(* CODESYS project Piezo.library
   Company: ESO
   Description: Local Device Control - LDC Piezo Library based on State Machine
   Version: 0.6.6.3
   Placeholder: ESO LDC Piezo Library
   Author: Dan Popovic
   Title: ESO LDC Piezo Library

Project tree, tasks and I/O mapping:
  libraries: Tc2_Standard, * (Beckhoff Automation GmbH); Tc2_System, * (Beckhoff Automation GmbH); Tc2_Utilities, * (Beckhoff Automation GmbH); Tc3_EventLogger, * (Beckhoff Automation GmbH); Tc3_Module, * (Beckhoff Automation GmbH); VisuDialogs, * (System); VisuSymbols, 3.5.10.0 (System)
  config/
    Device1_EtherCAT_SPLC014.xti
    Mappings_HW_SPLC014.xml
    Mappings_SIM.xml
  00000000-0000-0000-0000-000000000000|config\Device1_EtherCAT_SPLC014.xti
  00000000-0000-0000-0000-000000000000|config\Mappings_HW_SPLC014.xml
  00000000-0000-0000-0000-000000000000|config\Mappings_SIM.xml
  doc/
  DUTs/
    Enumerated/
      data type E_PIEZO_COMMAND
      data type E_PIEZO_ERROR
      data type E_PIEZO_EVENT
      data type E_PIEZO_HW_STATUS
      data type E_PIEZO_RPC_ERROR
      data type E_PIEZO_STATE
      data type E_PIEZO_STATUS
      data type E_PIEZO_SUBSTATE
    Structures/
      data type T_PIEZO_CFG
      data type T_PIEZO_CTRL
      data type T_PIEZO_DINT
      data type T_PIEZO_INFO
      data type T_PIEZO_INT
      data type T_PIEZO_LREAL
      data type T_PIEZO_STAT
      data type T_SIM_PIEZO_CFG
  GVLs/
    global variables GVL
  lib/
  POUs/
    Examples/
      function block FB_PIEZO_EXAMPLE [ST]: ActivityAuto, ActivityPos, M_Configure
    function block FB_PIEZO_BASE [ST]: ActionAutoExecute, ActionDisableExecute, ActionEnableExecute, ActionErrExecute, ActionHomeExecute, ActionInitExecute, ActionMaxOnFailure, ActionMoveBitExecute, ActionMoveUserExecute, ActionPosExecute, ActionResetExecute, ActionStopExecute, ActivityAuto, ActivityPos, CheckForEvents, M_CheckMaxOn, M_CheckRangeBit, M_CheckRangeUser, M_Configure, M_GetLogicalState, M_GetRpcErrorText, M_GetTimeInSec, M_LogEventDebug, M_LogEventEnd, M_LogEventError, M_LogEventGeneral, M_LogEventStart, M_ResetOutputs, M_RestartMaxOnTimer, M_SetRpcStatus, M_UpdateMonitor, ProcessEvents, RPC_Auto, RPC_Disable, RPC_Enable, RPC_Home, RPC_Init, RPC_MoveBit, RPC_MoveUser, RPC_Pos, RPC_Reset, RPC_SetDebug, RPC_SetLog, RPC_Stop, SetAction, SetEvent, SetHwStatus, SetLastCommand, SetState, SetStatus
    function block FB_SIM_PIEZO [ST]: RPC_ResetConfig, RPC_SetCouplerState, RPC_SetMaxError
    program MAIN [ST]
  Version/
    global variables Global_Version
  VISUs/
    Templates/
      visualisation GUI_TEMPLATE_PIEZO
    visualisation GUI_Piezo001
    visualisation GUI_Piezo002
  text list GlobalTextList
  00000000-0000-0000-0000-000000000000|Piezo.tmc
  Piezo.tmc
*)

// DUTs/Enumerated/E_PIEZO_COMMAND
{attribute 'qualified_only'}
{attribute 'strict'}
TYPE E_PIEZO_COMMAND :
(
	//
	// Events corresponding to commands
	// WARNING !!!
	// The values must be the same as in E_PIEZO_EVENT for E_PIEZO_COMMAND*, e.g.
	// EVENT_PIEZO_ENABLE = ENABLE
	//
	NONE	:= 0,
	
	RESET,
	INIT,
	STOP,
	ENABLE,
	DISABLE,
	AUTO,
	POS,
	HOME,
	MOVE_USER,
	MOVE_BIT
	
);
END_TYPE

// DUTs/Enumerated/E_PIEZO_ERROR
{attribute 'qualified_only'}
{attribute 'strict'}
TYPE E_PIEZO_ERROR :
(
	OK					:= 0,
	HW_NOT_OP,			
	ON_FAILURE,
	MAXON,
	OUT_OF_RANGE,
	USER2BIT_ZERO,
	
	// Simulator errors
	NOT_INITIALISED		:= 90,
	ZERO_POINTER		:= 100	
);
END_TYPE

// DUTs/Enumerated/E_PIEZO_EVENT
{attribute 'qualified_only'}
{attribute 'strict'}
TYPE E_PIEZO_EVENT :
(
	NONE	:= 0,
	
	//
	// Events corresponding to commands.
	// WARNING !!!
	// The values must be the same as in E_PIEZO_COMMAND for COMMAND_PIEZO_*, e.g.
	// ENABLE = COMMAND_PIEZO_ENABLE
	//
	RESET,
	INIT,
	STOP,
	ENABLE,
	DISABLE,
	AUTO,
	POS,
	HOME,
	MOVE_USER,
	MOVE_BIT,
	
	// 
	//	Events corresponding to internal events 
	//
	HWOK,
	ERRHW,
	ERRRANGE,
	ERRMAXON,
	ERRFAULT,
	ERRINIT,
	ERRDISABLE,
	USER2BIT_ZERO
	
);
END_TYPE

// DUTs/Enumerated/E_PIEZO_HW_STATUS
{attribute 'qualified_only'}
{attribute 'strict'}
TYPE E_PIEZO_HW_STATUS :
(
	UNKNOWN	:= 0,
	ERROR,
	ZERO,
	HOME,
	POS,
	AUTO
);
END_TYPE

// DUTs/Enumerated/E_PIEZO_RPC_ERROR
{attribute 'qualified_only'}
{attribute 'strict'}
TYPE E_PIEZO_RPC_ERROR :
(
	OK						:= 0,
	NOT_OP					:= -1,			
	NOT_NOTOP_READY			:= -2,			
	NOT_NOTOP_NOTREADY		:= -3,			
	LOCAL					:= -4,			
	MOVING_USER				:= -5,	// Out of limits target when moving in UU
	MOVING_BIT				:= -6	// Out of limits target when moving in bits			
);
END_TYPE

// DUTs/Enumerated/E_PIEZO_STATE
{attribute 'qualified_only'}
{attribute 'strict'}
TYPE E_PIEZO_STATE :
(
	NONE	:= 0,
	NOTOP,
	OP
);
END_TYPE

// DUTs/Enumerated/E_PIEZO_STATUS
{attribute 'qualified_only'}
{attribute 'strict'}
TYPE E_PIEZO_STATUS :
(
	OK	:= 0,
	ERROR
);
END_TYPE

// DUTs/Enumerated/E_PIEZO_SUBSTATE
{attribute 'qualified_only'}
{attribute 'strict'}
TYPE E_PIEZO_SUBSTATE :
(
	NONE				:= 0,
	
	NOTOP_NOTREADY		:= 100,
	NOTOP_READY			:= 101,
	NOTOP_ERROR			:= 199,
	
	OP_POS				:= 203,            
	OP_AUTO				:= 204,
	OP_ERROR			:= 299
);
END_TYPE

// DUTs/Structures/T_PIEZO_CFG
TYPE T_PIEZO_CFG :
STRUCT
	sName:			STRING	:= 'Piezo';	// Instance name
	nNumAxes:		INT := 3;		// Default 3 axes [0..2]

	nMaxOn:			DINT := 0;		// Maximum time for Piezo to be active [sec].
									// It goes to zero after this time.
									// If equal zero, check is not done.
									
	// Important note:
	// OPC UA cannot access individual items in arrays, e.g. nHome[2].
	// However, it can access, e.g. nHome[2].nValue.
	// That's why all configurable parameters are of type T_PIEZO_INT or T_PIEZO_LREAL.

	// Full range of A/D converter for analog output. Default is 15-bit.
	// Beckhoff 16-bit analog output terminals include the sign.
	// Effectively, for 0-10V terminals, this is a 15-bit resolution.
	nFullRange:		ARRAY [0..(GVL.C_nNumAxes-1)] OF T_PIEZO_INT;	// HOME position [bit]
	nHome:			ARRAY [0..(GVL.C_nNumAxes-1)] OF T_PIEZO_INT;	// HOME position [bit]
	nLimitLow:		ARRAY [0..(GVL.C_nNumAxes-1)] OF T_PIEZO_INT;	// Output lower limit [bit]
	nLimitHigh:		ARRAY [0..(GVL.C_nNumAxes-1)] OF T_PIEZO_INT;	// Output upper limit [bit]
	
	//
	// Conversions
	//
	// Conversion from User units (UU), i.e. Volts, to bits for SET values, i.e. OUTPUTS!
	// stat.nSetPosBit[i] := cfg.nUserOffsetBit_Set[i].nValue  +  stat.lrPosUsr[i] * cfg.lrUser2Bit[i].lrValue   (units [bit])
	//
	lrUser2Bit_Set:		ARRAY [0..(GVL.C_nNumAxes-1)] OF T_PIEZO_LREAL;	// Scale UU [V] to bits (default 10V=32767 bit)
	nUserOffsetBit_Set:	ARRAY [0..(GVL.C_nNumAxes-1)] OF T_PIEZO_INT;	// Offset [bit]

	//
	// Conversion from User units (UU), i.e. Volts, to bits for GET values, i.e. INPUTS, FEEDBACK!
	// stat.nActPosBit[i] := 
	//    cfg.nUserOffsetBit_Get[i].lrValue  +  stat.lrActPosUsr[i].lrValue * cfg.lrUser2Bit[i].lrValue   (units [bit])
	// stat.lrActPosUsr[i].lrValue := 
	//   (stat.nActPosBit[i].nValue - cfg.nUserOffsetBit_Get[i].nValue) / cfg.lrUser2Bit_Get[i].lrValue
	//
	lrUser2Bit_Get:		ARRAY [0..(GVL.C_nNumAxes-1)] OF T_PIEZO_LREAL;	// Scale UU [V] to bits (default 10V=32767 bit)
	nUserOffsetBit_Get:	ARRAY [0..(GVL.C_nNumAxes-1)] OF T_PIEZO_INT;	// Offset [bit]

	// Logging
	bLogExtTime:		BOOL 	:= FALSE;		// If TRUE, use external time in event logs. Default FALSE.
	bDebug:				BOOL 	:= FALSE;		// If TRUE, show event logs of Debug type. Default FALSE.
	bLog:				BOOL 	:= TRUE;		// If TRUE, log events. Default TRUE.
	
END_STRUCT
END_TYPE

// DUTs/Structures/T_PIEZO_CTRL
TYPE T_PIEZO_CTRL :
STRUCT
	nCommand:	E_PIEZO_COMMAND	:= E_PIEZO_COMMAND.NONE;			// See E_PIEZO_COMMAND
	bExecute:	BOOL;

	nPosBit:	ARRAY [0..(GVL.C_nNumAxes-1)] OF T_PIEZO_INT; 		// Set position in A/D Converter bits
	lrPosUser:	ARRAY [0..(GVL.C_nNumAxes-1)] OF T_PIEZO_LREAL; 	// Set position in user units
	
END_STRUCT
END_TYPE

// DUTs/Structures/T_PIEZO_DINT
TYPE T_PIEZO_DINT :
STRUCT
	nValue:	DINT;
END_STRUCT
END_TYPE

// DUTs/Structures/T_PIEZO_INFO
TYPE T_PIEZO_INFO :
STRUCT
(*
Driver Information 

Change Log:
	0.1	2017-07-17	- First version.
	0.2	2017-08-23	- Implemented suggestions from Luigi.
					- Implementation of HOME command.
					- POS command keep the piezos where they are.
	0.3	2017-09-05	- Cleanup.
					- Removed COMMAND_PIEZO_CONFIG and EVENT_PIEZO_CONFIG.
					- Removed COMMAND_PIEZO_MODE and EVENT_PIEZO_MODE.
					- Removed trg: R_TRIG.
					- Removed METHOD UpdateTimes.
					- Implemented MaxOn protection.
	0.4	2017-09-06	- Fully implemented RPC calls.
					- Cleanup of Status structure.
	0.5.0.0			- Extended to three axes.
					- Addition of library category ESO/ELT.
					- Tc2_System.F_GetSystemTime() used in M_GetTimeInSec().
	0.6.0.0	- Compiled with TC3.1.4022.25.
			- Renaming States STANDBY->NOTOP & FAILURE->ERROR.
	0.6.1.0	- Compiled with TC3.1.4022.27.
			- Cleaned code using Static Analysis tool.
			- Enumerated types are 'strict'.
			- Some enumerated types are set as type DINT.
			- Arrays start with zero index, i.e. [0..
			- Support of up to six axes (FB_PIEZO example is for three axes).
	0.6.1.1	- Cleanup.
			- Addition of logging.
	0.6.2.0	- Shortened enumerations.
	0.6.3.0	- Implemented RPC calls.
	0.6.4.0	- Moved whatever possible to FB_PIEZO_BASE.
			- Removed configuration arrays from input parameters.
			- Renamed FB_PIEZO to FB_PIEZO_EXAMPLE.
	0.6.5.0	- Implemented simulator.
			- Addition of HWOK event handling.
*)
	sDate:			STRING(32)	:= '2019-04-15';
	sDescription:	STRING(80) 	:= 'State Machine based Piezo controller';
	sName:			STRING(64)	:= 'FB_PIEZO';
	sPlatform:		STRING(32)	:= 'CoDeSys';
	sSynopsis:		STRING(64)	:= 'State Machine based Piezo controller';
	nVersionMajor:	DINT		:= 0;
	nVersionMinor:	DINT		:= 6;
END_STRUCT
END_TYPE

// DUTs/Structures/T_PIEZO_INT
TYPE T_PIEZO_INT :
STRUCT
	nValue:	INT;
END_STRUCT
END_TYPE

// DUTs/Structures/T_PIEZO_LREAL
TYPE T_PIEZO_LREAL :
STRUCT
	lrValue:	LREAL;
END_STRUCT
END_TYPE

// DUTs/Structures/T_PIEZO_STAT
TYPE T_PIEZO_STAT :
STRUCT
	bLocal:			BOOL	:= FALSE;						(* if TRUE, device operated from PLC GUI *)

	nLastCommand:	E_PIEZO_COMMAND		:= E_PIEZO_COMMAND.NONE;			(* Last command sent to the device *)

	nErrorCode: 	E_PIEZO_ERROR 		:= E_PIEZO_ERROR.OK;				(* Error code *)
	nHwStatus: 		E_PIEZO_HW_STATUS	:= E_PIEZO_HW_STATUS.UNKNOWN; 	(* HW status. See E_PIEZO_HW_STATUS *)
	nRpcErrorCode: 	E_PIEZO_RPC_ERROR 	:= E_PIEZO_RPC_ERROR.OK;		(* RPC Error code *)
	nStatus: 		E_PIEZO_STATUS		:= E_PIEZO_STATUS.OK; 			(* Device status *)
	nState:			E_PIEZO_STATE		:= E_PIEZO_STATE.NOTOP;
	nSubstate:		E_PIEZO_SUBSTATE	:= E_PIEZO_SUBSTATE.NOTOP_NOTREADY;
	

	sErrorText: 	STRING 	:= 'OK'; 						(* Error text *)
	sHwStatus: 		STRING 	:= 'UNKNOWN'; 					(* HW Status in textual form: 'UNKNOWN', 'ERROR', 'ON' or 'OFF' *)
	sLastCommand:	STRING	:= 'NONE';						(* Last command, as string, sent to the device *)
	sLibVersion:	STRING	:= 'UNKNOWN';					(* Library version as string, e.g. '1.2.0.0' *)
	sRpcErrorText: 	STRING 	:= 'OK'; 						(* RPC Error text *)
	sStatus: 		STRING 	:= 'OK'; 						(* Status in textual form, e.g. 'OFF' *)
	
	sState:			STRING	:= 'NOT OP';
	sSubstate:		STRING	:= 'NOT READY';
	
	sActionDesc:	STRING	:= '';
	sEventDesc:		STRING	:= '';
	
	nCycleCounter:	UDINT	:= 0;							// Alive flag
	nCycleTime:		UDINT	:= 0;							// Cycle time in us (microsec)

	lrSetPosUsr:	ARRAY [0..(GVL.C_nNumAxes-1)] OF T_PIEZO_LREAL; 	// Set position in user units
	lrActPosUsr:	ARRAY [0..(GVL.C_nNumAxes-1)] OF T_PIEZO_LREAL; 	// Actual position in user units
	nSetPosBit:		ARRAY [0..(GVL.C_nNumAxes-1)] OF T_PIEZO_INT; 		// Set position in ADC bits
	nActPosBit:		ARRAY [0..(GVL.C_nNumAxes-1)] OF T_PIEZO_DINT; 		// Actual position in ADC bits

	nTimeOn: 		UDINT 	:= 0;						// Time device has been active [sec] 
	
	// EICSSW-634: 
	// Slow updating OPC UA attributes to be monitored by the WS manager.
	// These attributes are updated every 100 ms.
	//
	
	// Number of cycles to skip to get update every 100 ms (default = 100 cycles).
	// Correctly set in M_Configure() taking into account cycle time.
	nMonSkipCycles:	DINT	:= 100;	
	
	monSetPosBit_0:	DINT;	// i.e. nSetPosBit[0].nValue
	monSetPosBit_1:	DINT;
	monSetPosBit_2:	DINT;
	monActPosBit_0:	DINT;	// i.e. nActPosBit[0].nValue
	monActPosBit_1:	DINT;
	monActPosBit_2:	DINT;
	monSetPosUsr_0:	LREAL;	// i.e. lrSetPosUsr[0].lrValue
	monSetPosUsr_1:	LREAL;
	monSetPosUsr_2:	LREAL;
	monActPosUsr_0:	LREAL;	// i.e. lrActPosUsr[0].lrValue
	monActPosUsr_1:	LREAL;
	monActPosUsr_2:	LREAL;

END_STRUCT
END_TYPE

// DUTs/Structures/T_SIM_PIEZO_CFG
TYPE T_SIM_PIEZO_CFG :
STRUCT
	nMaxError:		INT 	:= 0;		// Maximal Simulated feedback error [bit]
	nSignalCycle:	UDINT	:= 10000;	// Period for complete sine wave error cycle [msec] 
END_STRUCT
END_TYPE

// GVLs/GVL
{attribute 'qualified_only'}
VAR_GLOBAL CONSTANT
	{attribute 'OPC.UA.DA' := '0'}
	C_nNumAxes:	INT	:= 3;
END_VAR

// Version/Global_Version
{attribute 'TcGenerated'}
{attribute 'no-analysis'}
{attribute 'linkalways'}
// This function has been automatically generated from the project information.
VAR_GLOBAL CONSTANT
	{attribute 'const_non_replaced'}
	stLibVersion_ESO_LDC_Piezo_Library : ST_LibVersion := (iMajor := 0, iMinor := 6, iBuild := 6, iRevision := 3, nFlags := 0, sVersion := '0.6.6.3');
END_VAR

// POUs/Examples/FB_PIEZO_EXAMPLE
// Example of piezo with 3 axes
FUNCTION_BLOCK FB_PIEZO_EXAMPLE EXTENDS FB_PIEZO_BASE
VAR_INPUT
END_VAR
VAR_OUTPUT
END_VAR
VAR
	// NOTE: In this example we didn't extend any of the structures 
	//       but this could have been done.
	//    Example:
	//       T_PIEZO_CFG_EXAMPLE EXTENDS T_PIEZO_CFG
	//       cfg:	T_PIEZO_CFG_EXAMPLE;
	{attribute 'OPC.UA.DA' := '1'}
	cfg:		T_PIEZO_CFG;	
	{attribute 'OPC.UA.DA' := '1'}
	ctrl:		T_PIEZO_CTRL;	
	{attribute 'OPC.UA.DA' := '1'}
	{attribute 'OPC.UA.DA.Access' := '1'}
	stat:		T_PIEZO_STAT;	(* ReadOnly *)
	
	(***** Local variables *****)
	{attribute 'OPC.UA.DA' := '0'}
	nSetVal:		ARRAY [0..2] OF INT;	// Current set value [bit]
	{attribute 'OPC.UA.DA' := '0'}
	nLastCorr:		ARRAY [0..2] OF INT;	// Last correction [bit]
	{attribute 'OPC.UA.DA' := '0'}
	nScale:			ARRAY [0..2] OF INT := [1,1,1];	// +1 or -1 (going up or down)


END_VAR

// Set references !!! a MUST !!!
RefCfg	REF=cfg;
RefCtrl	REF=ctrl;
RefStat	REF=stat;

// Execute the base class object FB_LAMP_BASE
SUPER^();

METHOD ActivityAuto
VAR_INPUT
END_VAR
VAR
	i:	INT;
	nCorrection:	INT	:= 0;
	nNextVal:		INT	:= 0;
END_VAR
//
// This method should be overloaded by a User Method with specific behaviour.
//

// Add here code to automatically update piezo position.
// This is a dummy implementation where we want the following:
// Increment the output by 10 bits on every cycle.
// If upper limit is reached, start decrementing.
// If lower limit is reached, start incrementing.
// Ensure that the feedback reading equals the set value.
// To do this, the output might be slightly adjusted by the difference
// between the last set value and the actual value.

// Analog input channels as Int16
//  0 V = 0 bit
// 10 V = 32767 bit

// Don't move piezos if error is active.
IF stat.nErrorCode <> E_PIEZO_ERROR.OK THEN
	RETURN;
END_IF

FOR i:=0 TO cfg.nNumAxes-1 DO
	// Read feedback
	stat.nActPosBit[i].nValue	:= INT_TO_DINT(i_nActVal_Int16[i]);
	// Convert feedback to User Units [UU]
	IF cfg.lrUser2Bit_Get[i].lrValue <> 0.0 THEN
		stat.lrActPosUsr[i].lrValue := 
		   (stat.nActPosBit[i].nValue - cfg.nUserOffsetBit_Get[i].nValue) / cfg.lrUser2Bit_Get[i].lrValue;
	END_IF
	
	// Apply only small corrections.
	// The initial error could be huge and we want to avoid correcting it.
	IF ABS(nSetVal[i]) <> 32767 THEN
		nCorrection		:= 	nSetVal[i] - i_nActVal_Int16[i];
		IF ABS(nCorrection) < 100 THEN
			nLastCorr[i]	:= 	nCorrection;
		ELSE
			nLastCorr[i]	:= 	0;
		END_IF
	END_IF

	// nSetVal is the value we would like to get from the feedback
	nNextVal	:= nSetVal[i] + nScale[i]*10;
	IF ((nScale[i] = 1) AND (nNextVal >= cfg.nLimitHigh[i].nValue)) THEN	// overrun
		nSetVal[i] := cfg.nLimitHigh[i].nValue;
		nScale[i]	:= -1;
	ELSIF ((nScale[i] = -1) AND (nNextVal <= cfg.nLimitLow[i].nValue)) THEN
		nSetVal[i] := cfg.nLimitLow[i].nValue;
		nScale[i]	:= 1;
	ELSE
		nSetVal[i] := nNextVal;
	END_IF

	// Set the output that includes the correction in order to get i_nActVal[i] = nSetVal[i].
	q_nCtrl[i] := nSetVal[i] + nLastCorr[i];
	
		
	// Convert bits [bit] into user units [UU]
	stat.nSetPosBit[i].nValue		:=	q_nCtrl[i];
	IF cfg.lrUser2Bit_Set[i].lrValue <> 0.0 THEN
		stat.lrSetPosUsr[i].lrValue	:=	INT_TO_LREAL(q_nCtrl[i] - cfg.nUserOffsetBit_Set[i].nValue) / 
										cfg.lrUser2Bit_Set[i].lrValue;
	END_IF
END_FOR
END_METHOD

METHOD ActivityPos
VAR_INPUT
END_VAR
VAR
	i:	INT;
END_VAR
//
// This method should be overloaded by a User Method with specific behaviour.
//

// Dummy implementation.
// Update feedback
FOR i:=0 TO cfg.nNumAxes-1 DO
	// Read feedback
	stat.nActPosBit[i].nValue	:= INT_TO_DINT(i_nActVal_Int16[i]);
	// Convert feedback to User Units [UU]
	IF cfg.lrUser2Bit_Get[i].lrValue <> 0.0 THEN
		stat.lrActPosUsr[i].lrValue := 
		   (stat.nActPosBit[i].nValue - cfg.nUserOffsetBit_Get[i].nValue) / cfg.lrUser2Bit_Get[i].lrValue;
	END_IF
END_FOR
END_METHOD

METHOD M_Configure
VAR_INPUT
END_VAR
VAR
	i:	INT;
	fbGetCurTaskIdx:	GETCURTASKINDEX;
END_VAR
// If device is ready, there is nothing to configure.
IF bDeviceReady THEN
	RETURN;
END_IF

// TODO USER
// Customise the configuration starting from the COMPLETE FB_PIEZO_BASE::M_Configure().
// Modify the code between USER_START and USER_END

//
// USER_START
//

// If first cycle, copy configuration AND RETURN in order for the system to read all inputs before doing any work
IF stat.nCycleCounter = 0 THEN
	// Up to C_nNumAxes axes are supported
	// NOTE: In applications using Piezo.library, 
	//       GVL.C_nNumAxes has to be replaced with ESO_LDC_Piezo_Library.GVL.C_nNumAxes.
	IF in_nNumAxes > GVL.C_nNumAxes THEN
		cfg.nNumAxes	:= GVL.C_nNumAxes;
	ELSE
		cfg.nNumAxes	:=	in_nNumAxes;
	END_IF
	
	// Get cycle time in microsec.
	// CycleTime in _TaskInfo is given in 100 ns. 1 us = 1000 ns
	fbGetCurTaskIdx();	// Get the task index.
	RefStat.nCycleTime	:= TwinCAT_SystemInfoVarList._TaskInfo[fbGetCurTaskIdx.index].CycleTime/10;
	// Monitored attributes will change on every cycle, e.g. at 1 kHz.
	// In order to reduce load of OPC UA Server, update these attributes every 100 ms (100,000 us)
	RefStat.nMonSkipCycles	:= 100000 / UDINT_TO_DINT(RefStat.nCycleTime);
	
	// Hard code EXAMPLE configuration.
	// Note: Apart from the setting of cfg.nNumAxes, 
	//       the rest could be configured from the WS.
	// Note: The configuration can still be overwritten on INIT !!!

	// Assign input parameters to the configuration.
	cfg.sName		:=	in_sName;
	cfg.nMaxOn		:=	in_nMaxOn;	

	// Populate arrays in the configuration
	FOR i:= 0 TO (cfg.nNumAxes-1) DO
		cfg.nFullRange[i].nValue	:=	32767;
		cfg.nHome[i].nValue			:=	10 * i;	// Dummy value just to be <> 0
		cfg.nLimitLow[i].nValue		:=	100;
		cfg.nLimitHigh[i].nValue	:=	32500;
		//
		// Conversion from User units (UU) to [bit], e.g. [V] to [bit] for OUTPUTS
		// stat.nPosBit[i] := cfg.nUserOffset[i]  +  stat.lrPosUsr[i] * cfg.lrUser2Bit[i]   (units [bit])
		//
		cfg.lrUser2Bit_Set[i].lrValue		:=	3276.7;	// 1V = 3276.7 bits
		cfg.nUserOffsetBit_Set[i].nValue	:=	0;

		//
		// Conversion from User units (UU) to [bit], e.g. [V] to [bit] for INPUTS, i.e. feedback
		// stat.nPosBit[i] := cfg.nUserOffset[i]  +  stat.lrPosUsr[i] * cfg.lrUser2Bit[i]   (units [bit])
		//
		cfg.lrUser2Bit_Get[i].lrValue		:=	3276.7;	// 1V = 3276.7 bits
		cfg.nUserOffsetBit_Get[i].nValue	:=	0;
	END_FOR


	// Get the version number 
	stat.sLibVersion	:= stLibVersion_ESO_LDC_Piezo_Library.sVersion;

	// Increment counter.
	stat.nCycleCounter	:= stat.nCycleCounter + 1;
	RETURN;
ELSIF (stat.nCycleCounter * stat.nCycleTime) < 5000000 THEN
	// EtherCAT is normally ready after 3.5 sec.
	// We give it 5 sec to consider it to be ready.
	// Increment counter.
	stat.nCycleCounter	:= stat.nCycleCounter + 1;
	RETURN;
END_IF

//
// USER_END
//

// Don't touch the code below !!!

// After 100 cycles the system is ready, e.g. coupler state is 8.

// Create Event instances
fbEventStart.CreateEx	(TC_EVENTS.PiezoOpsEventClass.ActionStart,0);
fbEventEnd.CreateEx		(TC_EVENTS.PiezoOpsEventClass.ActionEnd,0);
fbEventError.CreateEx	(TC_EVENTS.PiezoOpsEventClass.Error,0);
fbEventDebug.CreateEx	(TC_EVENTS.PiezoOpsEventClass.Debug,0);
fbEventGeneral.CreateEx	(TC_EVENTS.PiezoOpsEventClass.General,0);

// The device is ready now.
bDeviceReady := TRUE;


// Clear errors
stat.nErrorCode		:= E_PIEZO_ERROR.OK;
stat.sErrorText		:= 'OK';
END_METHOD

END_FUNCTION_BLOCK

// POUs/FB_PIEZO_BASE
// Function Block for control of up to three analog outputs.
// The FB is intended for use with Piezo controllers.
FUNCTION_BLOCK FB_PIEZO_BASE
VAR_INPUT
	{attribute 'OPC.UA.DA' := '0'}
	in_sName:		STRING;			// Instance name. Default 'Piezo'.
	{attribute 'OPC.UA.DA' := '0'}
	in_nNumAxes:	INT;			// Max 3 axes

	{attribute 'OPC.UA.DA' := '0'}
	in_nMaxOn:		DINT	:= 0;	// Maximum time for Piezo to be active [sec].
									// Outputs go to zero after this time.
									// If equal zero, check is not done.
END_VAR
VAR_OUTPUT
END_VAR
VAR RETAIN
END_VAR
VAR
	{attribute 'OPC.UA.DA' := '0'}
	RefCfg:		REFERENCE TO T_PIEZO_CFG;	
	{attribute 'OPC.UA.DA' := '0'}
	RefCtrl:	REFERENCE TO T_PIEZO_CTRL;	
	{attribute 'OPC.UA.DA' := '1'}
	{attribute 'OPC.UA.DA.Access' := '1'}
	info:		T_PIEZO_INFO;	(* ReadOnly *)
	{attribute 'OPC.UA.DA' := '0'}
	{attribute 'OPC.UA.DA.Access' := '1'}
	RefStat:	REFERENCE TO T_PIEZO_STAT;	(* ReadOnly *)

	{attribute 'OPC.UA.DA' := '0'}
	nEvent:		      	DINT := E_PIEZO_EVENT.NONE;
	{attribute 'OPC.UA.DA' := '0'}
	nInternalEvent:		DINT := E_PIEZO_EVENT.NONE;
	
	// Operational Events
	{attribute 'OPC.UA.DA' := '0'}
	fbEventStart:	FB_TcMessage;
	{attribute 'OPC.UA.DA' := '0'}
	fbEventEnd:		FB_TcMessage;
	{attribute 'OPC.UA.DA' := '0'}
	fbEventError:	FB_TcMessage;
	{attribute 'OPC.UA.DA' := '0'}
	fbEventDebug:	FB_TcMessage;
	{attribute 'OPC.UA.DA' := '0'}
	fbEventGeneral:	FB_TcMessage;
	
	(***** Physical signals - to be mapped!!! *****)

	// Analog input channels as Int16 (might not exist)
	{attribute 'OPC.UA.DA' := '0'}
	i_nActVal_Int16	AT %I*: ARRAY [0..2] OF	INT;	// Control feedback, actual value

	// Analog input channels as Int32 (might not exist)
	{attribute 'OPC.UA.DA' := '0'}
	i_nActVal_Int32	AT %I*: ARRAY [0..2] OF	DINT;	// Control feedback, actual value

	(* Outputs *)
	{attribute 'OPC.UA.DA' := '0'}
	q_nCtrl 		AT %Q*: 	ARRAY [0..(GVL.C_nNumAxes-1)] OF	INT;	// Control analog output [bit]

	(* Inputs *)	
	{attribute 'OPC.UA.DA' := '0'}
	i_nCouplerState	AT %I*: 		UINT;	(* Link it to Coupler->InfoData->State *)

	// Flag if the device is ready to receive commands.
	// It takes a couple of cycles for the system to read inputs after reboot.
	{attribute 'OPC.UA.DA' := '0'}
	bDeviceReady:		BOOL 	:= FALSE;

	{attribute 'OPC.UA.DA' := '0'}
	toutMaxOn:	TON;
END_VAR

// On first cycle configure from input params and internally execute M_UserConfigure(), if exists.
IF NOT bDeviceReady THEN
	// Set device Configuration
	M_Configure();
	RETURN;
END_IF

// Increment counter.
// This will be seen as 'alive' flag.
RefStat.nCycleCounter	:= RefStat.nCycleCounter + 1;

// EICSSW-634:
M_UpdateMonitor();

(* === Check for commands and internal events to be processed === *)
CheckForEvents();

(* === Process events according to the State Machine === *)
ProcessEvents();

METHOD ActionAutoExecute
VAR_INPUT
END_VAR
SetAction('ActionAutoExecute');

// Log event
M_LogEventGeneral('AUTO mode activated');

// Restart safety timer
M_RestartMaxOnTimer();

(* Clear the error *)
SetStatus(E_PIEZO_ERROR.OK,'OK');

SetHwStatus(E_PIEZO_HW_STATUS.AUTO);
END_METHOD

METHOD ActionDisableExecute
VAR_INPUT
END_VAR
VAR
	i:	INT;
END_VAR
SetAction('ActionDisableExecute');

// Log event
M_LogEventGeneral('Device disabled');

// Zero the outputs
FOR i:=0 TO RefCfg.nNumAxes-1 DO
	q_nCtrl[i]					:=	0;	// bit
	RefStat.nSetPosBit[i].nValue		:=	q_nCtrl[i];
	IF RefCfg.lrUser2Bit_Set[i].lrValue <> 0.0 THEN
		RefStat.lrSetPosUsr[i].lrValue	:=	INT_TO_LREAL(q_nCtrl[i] - RefCfg.nUserOffsetBit_Set[i].nValue) / 
										RefCfg.lrUser2Bit_Set[i].lrValue;	// UU
	END_IF
END_FOR

SetHwStatus(E_PIEZO_HW_STATUS.ZERO);
END_METHOD

METHOD ActionEnableExecute
VAR_INPUT
END_VAR
VAR
	i:	INT;
END_VAR
SetAction('ActionEnableExecute');

// Log event
M_LogEventGeneral('Device enabled');

// Home the outputs
FOR i:=0 TO RefCfg.nNumAxes-1 DO
	q_nCtrl[i]			:= RefCfg.nHome[i].nValue;	// bit
	RefStat.nSetPosBit[i].nValue		:=	q_nCtrl[i];
	IF RefCfg.lrUser2Bit_Set[i].lrValue <> 0.0 THEN
		RefStat.lrSetPosUsr[i].lrValue	:=	INT_TO_LREAL(q_nCtrl[i] - RefCfg.nUserOffsetBit_Set[i].nValue) / 
										RefCfg.lrUser2Bit_Set[i].lrValue;	// UU
	END_IF
END_FOR

SetHwStatus(E_PIEZO_HW_STATUS.HOME);

(* Clear the error *)
SetStatus(E_PIEZO_ERROR.OK,'OK');
END_METHOD

METHOD ActionErrExecute
VAR
END_VAR
SetAction('ActionErrExecute');

IF nEvent = E_PIEZO_EVENT.ERRFAULT THEN
	RefStat.nErrorCode		:= E_PIEZO_ERROR.ON_FAILURE;
	RefStat.sErrorText		:= 'ERROR: Piezo HW failure';	
ELSIF nEvent = E_PIEZO_EVENT.ERRRANGE THEN
	RefStat.nErrorCode		:= E_PIEZO_ERROR.OUT_OF_RANGE;
	RefStat.sErrorText		:= 'ERROR: Piezo set position out of range';	
END_IF
		
RefStat.nStatus			:= E_PIEZO_STATUS.ERROR;
RefStat.sStatus			:= 'ERROR';
END_METHOD

METHOD ActionHomeExecute
VAR_INPUT
END_VAR
VAR
	i:	INT;
END_VAR
SetAction('ActionHomeExecute');

// Log event
M_LogEventGeneral('Actuators homed');

// Home the outputs
FOR i:=0 TO RefCfg.nNumAxes-1 DO
	q_nCtrl[i]					:=	RefCfg.nHome[i].nValue;	// bit
	RefStat.nSetPosBit[i].nValue		:=	q_nCtrl[i];
	IF RefCfg.lrUser2Bit_Set[i].lrValue <> 0.0 THEN
		RefStat.lrSetPosUsr[i].lrValue	:=	INT_TO_LREAL(q_nCtrl[i] - RefCfg.nUserOffsetBit_Set[i].nValue) / 
										RefCfg.lrUser2Bit_Set[i].lrValue;	// UU
	END_IF
END_FOR

// Restart safety timer
M_RestartMaxOnTimer();

SetHwStatus(E_PIEZO_HW_STATUS.HOME);

(* Clear the error *)
SetStatus(E_PIEZO_ERROR.OK,'OK');
END_METHOD

METHOD ActionInitExecute
VAR_INPUT
END_VAR
VAR
	i:	INT;
END_VAR
SetAction('ActionInitExecute');

// Log event
M_LogEventGeneral('Device initialised');

// Zero the outputs
FOR i:=0 TO RefCfg.nNumAxes-1 DO
	// Prevent division by zero due to wrong configuration
	IF RefCfg.lrUser2Bit_Set[i].lrValue = 0.0 THEN
		nEvent	:= E_PIEZO_EVENT.USER2BIT_ZERO;
		SetStatus(E_PIEZO_ERROR.USER2BIT_ZERO,'ERROR: cfg.lrUser2Bit has zero value.');
		RETURN;
	END_IF
	q_nCtrl[i]					:=	0;
	RefStat.nSetPosBit[i].nValue		:=	q_nCtrl[i];
	IF RefCfg.lrUser2Bit_Set[i].lrValue <> 0.0 THEN
		RefStat.lrSetPosUsr[i].lrValue	:=	INT_TO_LREAL(q_nCtrl[i] - RefCfg.nUserOffsetBit_Set[i].nValue) / 
										RefCfg.lrUser2Bit_Set[i].lrValue;	// UU
	END_IF
END_FOR

SetHwStatus(E_PIEZO_HW_STATUS.ZERO);

// Status OK 
SetStatus(E_PIEZO_ERROR.OK,'OK');
END_METHOD

METHOD ActionMaxOnFailure
VAR_INPUT
END_VAR
(* code to initiate the switching OFF of the lamp *)
SetAction('ActionMaxOnFailure');

// Log event
M_LogEventError('Max ON time exceeded. Actuators zeroed.');

(* Set the error *)
SetStatus(E_PIEZO_ERROR.MAXON,'ERROR: Maximum ON time exceeded.');
END_METHOD

METHOD ActionMoveBitExecute
VAR_INPUT
END_VAR
VAR
	i:	INT;
END_VAR
SetAction('ActionMoveBitExecute');

// Log event
M_LogEventGeneral('Actuators moved in [bit] units');

// Check if the positions are inside the allowed range
FOR i:=0 TO RefCfg.nNumAxes-1 DO
	IF NOT M_CheckRangeBit(nIndex:= i, nVal:= RefCtrl.nPosBit[i].nValue) THEN
		M_LogEventError('Set bit value out of range');
		nInternalEvent	:= E_PIEZO_EVENT.ERRRANGE;
//		SetEvent(E_PIEZO_EVENT.ERRRANGE);
		RETURN;
	END_IF
END_FOR


// Activate outputs
FOR i:=0 TO RefCfg.nNumAxes-1 DO
	q_nCtrl[i]			:= RefCtrl.nPosBit[i].nValue;
	RefStat.nSetPosBit[i].nValue		:=	q_nCtrl[i];
	IF RefCfg.lrUser2Bit_Set[i].lrValue <> 0.0 THEN
		RefStat.lrSetPosUsr[i].lrValue	:=	INT_TO_LREAL(q_nCtrl[i] - RefCfg.nUserOffsetBit_Set[i].nValue) / 
										RefCfg.lrUser2Bit_Set[i].lrValue;
	END_IF
END_FOR

// Restart safety timer
M_RestartMaxOnTimer();

SetHwStatus(E_PIEZO_HW_STATUS.POS);

// Status OK 
SetStatus(E_PIEZO_ERROR.OK,'OK');
END_METHOD

// Action to move piezos to specified User Position.
METHOD ActionMoveUserExecute
VAR_INPUT
END_VAR
VAR
	i:	INT;
END_VAR
SetAction('ActionMoveUserExecute');

// Log event
M_LogEventGeneral('Actuators moved in [UU] (user)  units');

// Check if the positions are inside the allowed range.
// If any position is out of range, don't set outputs.
FOR i:=0 TO RefCfg.nNumAxes-1 DO
	IF NOT M_CheckRangeUser(nIndex:= i, lrVal:= RefCtrl.lrPosUser[i].lrValue) THEN
		M_LogEventError('Set User value out of range');
		nInternalEvent	:= E_PIEZO_EVENT.ERRRANGE;
		RETURN;
	END_IF
END_FOR

// Set the outputs
FOR i:=0 TO RefCfg.nNumAxes-1 DO
	// Calculate the output [bit] including the offset
	q_nCtrl[i]	:= RefCfg.nUserOffsetBit_Set[i].nValue  +  LREAL_TO_INT(RefCtrl.lrPosUser[i].lrValue * RefCfg.lrUser2Bit_Set[i].lrValue);
	
	// Update the status in both [bit] and [UU]
	RefStat.nSetPosBit[i].nValue		:= q_nCtrl[i];
	RefStat.lrSetPosUsr[i].lrValue	:= RefCtrl.lrPosUser[i].lrValue;
END_FOR

// Restart safety timer
M_RestartMaxOnTimer();

SetHwStatus(E_PIEZO_HW_STATUS.POS);

// Status OK 
SetStatus(E_PIEZO_ERROR.OK,'OK');
END_METHOD

METHOD ActionPosExecute
VAR_INPUT
END_VAR
SetAction('ActionPosExecute');

// Log event
M_LogEventGeneral('Actuators stopped at current position');

// Restart safety timer
M_RestartMaxOnTimer();

// This action is normally called when exiting, i.e. stopping, AUTO mode.
// There is nothing to be done. Just keep current position.
SetHwStatus(E_PIEZO_HW_STATUS.POS);


(* Clear the error *)
SetStatus(E_PIEZO_ERROR.OK,'OK');
END_METHOD

METHOD ActionResetExecute
VAR_INPUT
END_VAR
SetAction('ActionResetExecute');

// Log event
M_LogEventGeneral('Device reset');

M_ResetOutputs(TRUE);
END_METHOD

METHOD ActionStopExecute
VAR_INPUT
END_VAR
SetAction('ActionStopExecute');

M_ResetOutputs(TRUE);
END_METHOD

METHOD ActivityAuto
VAR_INPUT
END_VAR
END_METHOD

METHOD ActivityPos
VAR_INPUT
END_VAR
END_METHOD

METHOD CheckForEvents
VAR_INPUT
END_VAR

(* 
	Start assuming the HW is OK. 
	This is needed to recover from the situation where 
	the HW was failing and now it is working.
*)
nEvent := E_PIEZO_EVENT.HWOK;


// Check if the piezo should be switched off for protection of HW.
M_CheckMaxOn();


(* 
	Check for events in the following order: 
   	1) HW failure: without HW avilability there is no point to do anything
	2) Internal events: to allow completing the initiated commands before 
                        starting processing new commands. 
   	3) Commands: to react to external commands. Commands should be executed 
                 before processing HW signals to allow to start a recovery action.
   	4) HW signals:  such as Lamp is ON/OFF.
*)

IF i_nCouplerState <> 8 THEN	
	(* Check if the HW is NOT OK *)
	(*
	If the hardware status is NOT OK, we cannot trust the readings.
	Variable i_nCouplerState has to be mapped to a State of a terminal, e.g. EK1100.
	The value should be 8.
 	*)
	SetEvent(E_PIEZO_EVENT.ERRHW);
	SetStatus(E_PIEZO_ERROR.HW_NOT_OP, 'ERROR: HW not in OPERATIONAL state');

ELSIF nInternalEvent <> E_PIEZO_EVENT.NONE THEN
	(* Handle internal events *)
	SetEvent(nInternalEvent);
	nInternalEvent := E_PIEZO_EVENT.NONE;
ELSIF RefCtrl.bExecute  THEN
	(* Handle commands *)
	RefCtrl.bExecute		:= FALSE;			(* Clear the Execute bit *)
	SetLastCommand(RefCtrl.nCommand);			(* Save the last command *)
	SetEvent(RefCtrl.nCommand);
	RefCtrl.nCommand 		:= E_PIEZO_COMMAND.NONE;	(* Clear the Command *)
END_IF
END_METHOD

METHOD M_CheckMaxOn
VAR_INPUT
END_VAR
VAR
	i:		INT;
	active:	BOOL	:= FALSE;
END_VAR
// Check if control is active, i.e. if there is any voltage applied.
// This means that one or more outputs are not zero [bit].
FOR i:=0 TO RefCfg.nNumAxes-1 DO
	IF q_nCtrl[i] <> 0 THEN
		active	:= TRUE;
	END_IF
END_FOR

// Do the check only if configured to do so.
IF RefCfg.nMaxOn <> 0 THEN
	toutMaxOn();	// Execute the timer with last settings
	IF active THEN
		// Restart the timer, if not running yet.
		IF TIME_TO_UDINT(toutMaxOn.ET) = 0 THEN
			// The timer is not running.
			// Restart the command timer
			toutMaxOn(IN:=FALSE);
			toutMaxOn(IN:=TRUE,PT:=DINT_TO_TIME(RefCfg.nMaxOn * 1000));
		END_IF
		toutMaxOn(IN:=TRUE,PT:=DINT_TO_TIME(RefCfg.nMaxOn * 1000));
		RefStat.nTimeOn	:= TIME_TO_UDINT(toutMaxOn.ET) / 1000;	// ms -> sec
	ELSE
		toutMaxOn(IN:=FALSE);	// Stop the timer
		RefStat.nTimeOn	:= 0;
	END_IF
	
	// Check if the timer expired, i.e. the output should be set to zero.
	IF toutMaxOn.Q THEN
		toutMaxOn(IN:=FALSE);	// Stop the timer
		M_ResetOutputs(FALSE);	// Reset (zero) all outputs, keep error.
		// This error set is needed in order to stop ActivityAuto updating positions.
		SetStatus(E_PIEZO_ERROR.MAXON,'ERROR: Maximum ON time exceeded.');
		nInternalEvent := E_PIEZO_EVENT.ERRMAXON;
	END_IF
ELSE
	// Check for MaxOn is not done.
	toutMaxOn(IN:=FALSE);	// Stop the timer
	RefStat.nTimeOn	:= 0;
	RETURN;
END_IF
END_METHOD

// Check if the value is inside lower and upper limits.
// Return TRUE if OK, otherwise FALSE.
METHOD M_CheckRangeBit : BOOL
VAR_INPUT
	nIndex:	INT;
	nVal:	INT;
END_VAR
IF nVal > RefCfg.nLimitHigh[nIndex].nValue THEN
	M_CheckRangeBit	:= FALSE;
ELSIF nVal < RefCfg.nLimitLow[nIndex].nValue THEN
	M_CheckRangeBit	:= FALSE;
ELSE
	M_CheckRangeBit	:= TRUE;	// OK
END_IF
END_METHOD

METHOD M_CheckRangeUser : BOOL
VAR_INPUT
	nIndex:	INT;
	lrVal:	LREAL;
END_VAR
VAR
	nTmpVal:	DINT;
END_VAR
// Get the value as DINT and check if AD converter limits are exceeded.
nTmpVal	:=	INT_TO_DINT(RefCfg.nUserOffsetBit_Set[nIndex].nValue)  +  
			LREAL_TO_DINT(lrVal * RefCfg.lrUser2Bit_Set[nIndex].lrValue);


IF nTmpVal > INT_TO_DINT(RefCfg.nLimitHigh[nIndex].nValue) THEN
	M_CheckRangeUser	:= FALSE;
ELSIF nTmpVal < INT_TO_DINT(RefCfg.nLimitLow[nIndex].nValue) THEN
	M_CheckRangeUser	:= FALSE;
ELSE
	M_CheckRangeUser	:= TRUE;
END_IF
END_METHOD

METHOD M_Configure
VAR_INPUT
END_VAR
VAR
	i:	INT;
	fbGetCurTaskIdx:	GETCURTASKINDEX;
END_VAR
// If device is ready, there is nothing to configure.
IF bDeviceReady THEN
	RETURN;
END_IF

// TODO USER
// Customise the configuration starting from the COMPLETE FB_PIEZO_BASE::M_Configure().
// Modify the code between USER_START and USER_END

//
// USER_START
//

// If first cycle, copy configuration AND RETURN in order for the system 
// to read all inputs before doing any work.
IF RefStat.nCycleCounter = 0 THEN
	// Up to C_nNumAxes axes are supported
	IF in_nNumAxes > GVL.C_nNumAxes THEN
		RefCfg.nNumAxes	:=	GVL.C_nNumAxes;
	ELSE
		RefCfg.nNumAxes	:=	in_nNumAxes;
	END_IF
	
	// Get cycle time in microsec.
	// CycleTime in _TaskInfo is given in 100 ns. 1 us = 1000 ns
	fbGetCurTaskIdx();	// Get the task index.
	RefStat.nCycleTime	:= TwinCAT_SystemInfoVarList._TaskInfo[fbGetCurTaskIdx.index].CycleTime/10;
	// Monitored attributes will change on every cycle, e.g. at 1 kHz.
	// In order to reduce load of OPC UA Server, update these attributes every 100 ms (100,000 us)
	RefStat.nMonSkipCycles	:= 100000 / UDINT_TO_DINT(RefStat.nCycleTime);
	
	// Hard code EXAMPLE configuration.
	// Note: Apart from the setting of cfg.nNumAxes, 
	//       the rest could be configured from the WS.
	// Note: The configuration can still be overwritten on INIT !!!

	// Assign input parameters to the configuration.
	RefCfg.sName		:=	in_sName;
	RefCfg.nMaxOn		:=	in_nMaxOn;	

	// Populate arrays in the configuration
	FOR i:= 0 TO (RefCfg.nNumAxes-1) DO
		RefCfg.nFullRange[i].nValue	:=	 32767;
		RefCfg.nHome[i].nValue			:=	0;
		RefCfg.nLimitLow[i].nValue		:=	-32767;
		RefCfg.nLimitHigh[i].nValue	:=	 32767;
		//
		// Conversion from User units (UU) to [bit], e.g. [V] to [bit] for OUTPUTS
		// stat.nPosBit[i] := cfg.nUserOffset[i]  +  stat.lrPosUsr[i] * cfg.lrUser2Bit[i]   (units [bit])
		//
		RefCfg.lrUser2Bit_Set[i].lrValue		:=	3276.7;	// 1V = 3276.7 bits
		RefCfg.nUserOffsetBit_Set[i].nValue	:=	0;

		//
		// Conversion from User units (UU) to [bit], e.g. [V] to [bit] for INPUTS, i.e. feedback
		// stat.nPosBit[i] := cfg.nUserOffset[i]  +  stat.lrPosUsr[i] * cfg.lrUser2Bit[i]   (units [bit])
		//
		RefCfg.lrUser2Bit_Get[i].lrValue		:=	3276.7;	// 1V = 3276.7 bits
		RefCfg.nUserOffsetBit_Get[i].nValue	:=	0;
	END_FOR


	// Get the version number 
	RefStat.sLibVersion	:= stLibVersion_ESO_LDC_Piezo_Library.sVersion;

	// Increment counter.
	RefStat.nCycleCounter	:= RefStat.nCycleCounter + 1;
	RETURN;
ELSIF (RefStat.nCycleCounter * RefStat.nCycleTime) < 5000000 THEN
	// EtherCAT is normally ready after 3.5 sec.
	// We give it 5 sec to consider it to be ready.
	// Increment counter.
	RefStat.nCycleCounter	:= RefStat.nCycleCounter + 1;
	RETURN;
END_IF

//
// USER_END
//

// Don't touch the code below !!!

// After 5 sec the system is ready, e.g. coupler state is 8.

// Create Event instances
fbEventStart.CreateEx	(TC_EVENTS.PiezoOpsEventClass.ActionStart,0);
fbEventEnd.CreateEx		(TC_EVENTS.PiezoOpsEventClass.ActionEnd,0);
fbEventError.CreateEx	(TC_EVENTS.PiezoOpsEventClass.Error,0);
fbEventDebug.CreateEx	(TC_EVENTS.PiezoOpsEventClass.Debug,0);
fbEventGeneral.CreateEx	(TC_EVENTS.PiezoOpsEventClass.General,0);

// The device is ready now.
bDeviceReady := TRUE;


// Clear errors
RefStat.nErrorCode		:= E_PIEZO_ERROR.OK;
RefStat.sErrorText		:= 'OK';
END_METHOD

METHOD M_GetLogicalState : BOOL
(*
	This method returns the state of the variable based on its 
	activeLow configuration.
	Syntax:
		bState	:= GetLogicalState (<var value>,  <activeLow cfg>);
		
	Example 1:
		var = TRUE;
		activeLow = FALSE;
		bState	:= GetLogicalState (TRUE,  FALSE); = TRUE

	Example 2:
		var = TRUE;
		activeLow = TRUE;
		bState	:= GetLogicalState (TRUE,  TRUE); = FALSE
*)
VAR_INPUT
	state:		BOOL;
	activeLow:	BOOL;
END_VAR
IF activeLow THEN
	M_GetLogicalState := NOT state;
ELSE
	M_GetLogicalState := state;
END_IF
END_METHOD

METHOD M_GetRpcErrorText : STRING
VAR_INPUT
	ErrorCode:	INT;
END_VAR
VAR
	str:	STRING;
END_VAR
CASE ErrorCode OF
	E_PIEZO_RPC_ERROR.OK:						str	:= 'OK';
	E_PIEZO_RPC_ERROR.NOT_OP:					str	:= 'Cannot control device. Not in OP state.';
	E_PIEZO_RPC_ERROR.NOT_NOTOP_READY:			str	:= 'Call failed. Not in NOTOP_READY.';
	E_PIEZO_RPC_ERROR.NOT_NOTOP_NOTREADY:		str	:= 'Call failed. Not in NOTOP_NOTREADY/ERROR.';
	E_PIEZO_RPC_ERROR.LOCAL:					str	:= 'RPC calls not allowed in Local mode.';
	E_PIEZO_RPC_ERROR.MOVING_USER:				str	:= 'Set user value out of range.';
	E_PIEZO_RPC_ERROR.MOVING_BIT:				str	:= 'Set bit value out of range.';
ELSE
	str	:= 'Unregistered RPC error.';
END_CASE

M_GetRpcErrorText	:= str;
END_METHOD

(*
	This method returns absolute time rounded to seconds.
*)
METHOD M_GetTimeInSec : UDINT
VAR_INPUT
END_VAR
VAR
END_VAR
// System time is given in 100ns. Divide by 10000000 to get in seconds. 
M_GetTimeInSec	:= ULINT_TO_UDINT(Tc2_System.F_GetSystemTime() / 10000000);
END_METHOD

METHOD M_LogEventDebug
VAR_INPUT
	sText:	STRING	:= '';
END_VAR
// Log Debug events only if both logging and debugging is enabled
IF  RefCfg.bLog AND RefCfg.bDebug THEN
	fbEventDebug.ipArguments.Clear().AddString(sText);
	fbEventDebug.Send(0);
END_IF
END_METHOD

METHOD M_LogEventEnd
VAR_INPUT
	sText:	STRING	:= '';
END_VAR
// Log only if logging is enabled
IF  NOT RefCfg.bLog THEN
	RETURN;
END_IF

fbEventEnd.ipArguments.Clear().AddString(sText);
fbEventEnd.Send(0);
END_METHOD

METHOD M_LogEventError
VAR_INPUT
	sText:	STRING	:= '';
END_VAR
// Log only if logging is enabled
IF  NOT RefCfg.bLog THEN
	RETURN;
END_IF

fbEventError.ipArguments.Clear().AddString(sText);
fbEventError.Send(0);
END_METHOD

METHOD M_LogEventGeneral
VAR_INPUT
	sText:	STRING	:= '';
END_VAR
// Log only if logging is enabled
IF  NOT RefCfg.bLog THEN
	RETURN;
END_IF

fbEventGeneral.ipArguments.Clear().AddString(sText);
fbEventGeneral.Send(0);
END_METHOD

METHOD M_LogEventStart
VAR_INPUT
	sText:	STRING	:= '';
END_VAR
// Log only if logging is enabled
IF  NOT RefCfg.bLog THEN
	RETURN;
END_IF

fbEventStart.ipArguments.Clear().AddString(sText);
fbEventStart.Send(0);
END_METHOD

METHOD M_ResetOutputs
VAR_INPUT
	in_bClearError:	BOOL := TRUE;
END_VAR
VAR
	i:	int;
END_VAR
(* Set piezo outputs to zero bits *)
FOR i:= 0 TO RefCfg.nNumAxes-1 DO
	q_nCtrl[i] := 0;
	RefStat.nSetPosBit[i].nValue		:=	q_nCtrl[i];
		IF RefCfg.lrUser2Bit_Set[i].lrValue <> 0.0 THEN
			RefStat.lrSetPosUsr[i].lrValue	:=	INT_TO_LREAL(q_nCtrl[i] - RefCfg.nUserOffsetBit_Set[i].nValue) / 
											RefCfg.lrUser2Bit_Set[i].lrValue;
		END_IF
END_FOR

IF in_bClearError THEN
	// Status OK 
	SetStatus(E_PIEZO_ERROR.OK, 'OK');
END_IF

SetHwStatus(E_PIEZO_HW_STATUS.ZERO);
END_METHOD

METHOD M_RestartMaxOnTimer
VAR_INPUT
END_VAR
VAR
	i:		INT;
	active:	BOOL	:= FALSE;
END_VAR
// Check if control is active, i.e. if there is any voltage applied.
// This means that one or more outputs are not zero [bit].
FOR i:=0 TO RefCfg.nNumAxes-1 DO
	IF q_nCtrl[i] <> 0 THEN
		active	:= TRUE;
	END_IF
END_FOR

// Do the check only if configured to do so,
// i.e. nMaxOn <> 0.
IF RefCfg.nMaxOn <> 0 THEN
	toutMaxOn();	// Execute the timer with last settings
	IF active THEN
		toutMaxOn(IN:=FALSE);
		toutMaxOn(IN:=TRUE,PT:=DINT_TO_TIME(RefCfg.nMaxOn * 1000));
		RefStat.nTimeOn	:= 0;
	ELSE
		toutMaxOn(IN:=FALSE);	// Stop the timer
		RefStat.nTimeOn	:= 0;
	END_IF
END_IF
END_METHOD

METHOD M_SetRpcStatus : INT
VAR_INPUT
	nErrorCode:	E_PIEZO_RPC_ERROR;
END_VAR
RefStat.nRpcErrorCode	:= nErrorCode;
RefStat.sRpcErrorText	:= M_GetRpcErrorText(nErrorCode);

M_SetRpcStatus		:= nErrorCode;
END_METHOD

METHOD M_UpdateMonitor
VAR_INPUT
END_VAR
// Update monitored attributes every RefStat.nMonSkipCycles
IF UDINT_TO_DINT(RefStat.nCycleCounter) MOD RefStat.nMonSkipCycles = 0 THEN
	RefStat.monSetPosBit_0	:= RefStat.nSetPosBit[0].nValue;
	RefStat.monSetPosBit_1	:= RefStat.nSetPosBit[1].nValue;
	RefStat.monSetPosBit_2	:= RefStat.nSetPosBit[2].nValue;
	
	RefStat.monActPosBit_0	:= RefStat.nActPosBit[0].nValue;
	RefStat.monActPosBit_1	:= RefStat.nActPosBit[1].nValue;
	RefStat.monActPosBit_2	:= RefStat.nActPosBit[2].nValue;
	
	RefStat.monSetPosUsr_0	:= RefStat.lrSetPosUsr[0].lrValue;
	RefStat.monSetPosUsr_1	:= RefStat.lrSetPosUsr[1].lrValue;
	RefStat.monSetPosUsr_2	:= RefStat.lrSetPosUsr[2].lrValue;
	
	RefStat.monActPosUsr_0	:= RefStat.lrActPosUsr[0].lrValue;
	RefStat.monActPosUsr_1	:= RefStat.lrActPosUsr[1].lrValue;
	RefStat.monActPosUsr_2	:= RefStat.lrActPosUsr[2].lrValue;
END_IF
END_METHOD

METHOD ProcessEvents
VAR_INPUT
END_VAR

VAR
END_VAR

(* 
	Before processing the event, execute the Do-Activity tasks. 
	Note that, in case of orthogonal regions, more than one Do-Activity 
	could run in the same PLC cycle.
	Note: Most of these activities have timeouts since they take time.
*)


IF RefStat.nSubstate = E_PIEZO_SUBSTATE.OP_AUTO THEN
	ActivityAuto();	// Just update times
END_IF

IF RefStat.nSubstate = E_PIEZO_SUBSTATE.OP_POS THEN
	ActivityPos();	// Just update times
END_IF



(* 
	Evaluate state machine transitions.
*)

CASE RefStat.nState OF

//***********************************
// NOTOP
//***********************************
E_PIEZO_STATE.NOTOP:

	(* Transitions from NOTOP substates *)
	CASE RefStat.nSubstate OF
	
	E_PIEZO_SUBSTATE.NOTOP_NOTREADY:		
		IF nEvent = E_PIEZO_EVENT.RESET THEN
			ActionResetExecute();
			RETURN;
		ELSIF nEvent = E_PIEZO_EVENT.INIT THEN
			ActionInitExecute();
			// ActionInitExecute() might set nEvent to E_PIEZO_EVENT.USER2BIT_ZERO
			// in case of wrong configuration.
			// If nEvent has changed, something is wrong.
			IF nEvent = E_PIEZO_EVENT.INIT THEN
				// Nothing has changed, all OK.
				SetState(E_PIEZO_STATE.NOTOP, E_PIEZO_SUBSTATE.NOTOP_READY);
			ELSE
				SetState(E_PIEZO_STATE.NOTOP, E_PIEZO_SUBSTATE.NOTOP_ERROR);
			END_IF
			RETURN;
		END_IF
		
	E_PIEZO_SUBSTATE.NOTOP_READY:			
		IF nEvent = E_PIEZO_EVENT.RESET THEN
			ActionResetExecute();
			SetState(E_PIEZO_STATE.NOTOP, E_PIEZO_SUBSTATE.NOTOP_NOTREADY);
			RETURN;
		ELSIF nEvent = E_PIEZO_EVENT.ERRFAULT THEN
			SetState(E_PIEZO_STATE.NOTOP, E_PIEZO_SUBSTATE.NOTOP_NOTREADY);			
			RETURN;
		ELSIF nEvent = E_PIEZO_EVENT.ERRMAXON THEN
			ActionMaxOnFailure();
			RETURN;				
		ELSIF nEvent = E_PIEZO_EVENT.ENABLE THEN
			ActionEnableExecute();
			SetState(E_PIEZO_STATE.OP, E_PIEZO_SUBSTATE.OP_POS);
			RETURN;
		ELSIF nEvent = E_PIEZO_EVENT.STOP THEN
			ActionStopExecute();
			RETURN;
		END_IF

	E_PIEZO_SUBSTATE.NOTOP_ERROR:			
		IF nEvent = E_PIEZO_EVENT.HWOK THEN
			SetState(E_PIEZO_STATE.NOTOP, E_PIEZO_SUBSTATE.NOTOP_NOTREADY);
			RETURN;
		END_IF
		
	END_CASE

	(* Transitions from NOTOP state *)
	IF nEvent = E_PIEZO_EVENT.ERRHW THEN
		SetState(E_PIEZO_STATE.NOTOP, E_PIEZO_SUBSTATE.NOTOP_ERROR);
		RETURN;
	END_IF
	
//***********************************
// OPERATIONAL
//***********************************
E_PIEZO_STATE.OP:

	(* Transitions from OP substates *)
	CASE RefStat.nSubstate OF
	E_PIEZO_SUBSTATE.OP_POS:			
		IF nEvent = E_PIEZO_EVENT.POS THEN
			ActionPosExecute();
			RETURN;
		ELSIF nEvent = E_PIEZO_EVENT.HOME THEN
			ActionHomeExecute();
			RETURN;
		ELSIF nEvent = E_PIEZO_EVENT.AUTO THEN
			ActionAutoExecute();
			SetState(E_PIEZO_STATE.OP, E_PIEZO_SUBSTATE.OP_AUTO);
			RETURN;
		ELSIF nEvent = E_PIEZO_EVENT.DISABLE THEN
			ActionDisableExecute();
			SetState(E_PIEZO_STATE.NOTOP, E_PIEZO_SUBSTATE.NOTOP_READY);
			RETURN;		
		ELSIF nEvent = E_PIEZO_EVENT.MOVE_BIT THEN
			ActionMoveBitExecute();
			RETURN;	
		ELSIF nEvent = E_PIEZO_EVENT.MOVE_USER THEN
			ActionMoveUserExecute();
			RETURN;	
		ELSIF nEvent = E_PIEZO_EVENT.ERRFAULT THEN
			ActionErrExecute();
			SetState(E_PIEZO_STATE.OP, E_PIEZO_SUBSTATE.OP_ERROR);
			RETURN;				
		ELSIF nEvent = E_PIEZO_EVENT.ERRRANGE THEN
			ActionErrExecute();
			SetState(E_PIEZO_STATE.OP, E_PIEZO_SUBSTATE.OP_ERROR);
			RETURN;				
		ELSIF nEvent = E_PIEZO_EVENT.ERRMAXON THEN
			ActionMaxOnFailure();
			SetState(E_PIEZO_STATE.OP, E_PIEZO_SUBSTATE.OP_ERROR);
			RETURN;				
		ELSIF nEvent = E_PIEZO_EVENT.STOP THEN
			ActionStopExecute();
			RETURN;
		END_IF

	E_PIEZO_SUBSTATE.OP_AUTO:			
		IF nEvent = E_PIEZO_EVENT.POS THEN
			ActionPosExecute();
			SetState(E_PIEZO_STATE.OP, E_PIEZO_SUBSTATE.OP_POS);
			RETURN;
		ELSIF nEvent = E_PIEZO_EVENT.HOME THEN
			ActionHomeExecute();
			SetState(E_PIEZO_STATE.OP, E_PIEZO_SUBSTATE.OP_POS);
			RETURN;
		ELSIF nEvent = E_PIEZO_EVENT.AUTO THEN
			ActionAutoExecute();
			RETURN;
		ELSIF nEvent = E_PIEZO_EVENT.DISABLE THEN
			ActionDisableExecute();
			SetState(E_PIEZO_STATE.NOTOP, E_PIEZO_SUBSTATE.NOTOP_READY);
			RETURN;	
		ELSIF nEvent = E_PIEZO_EVENT.MOVE_BIT THEN
			ActionMoveBitExecute();
			SetState(E_PIEZO_STATE.OP, E_PIEZO_SUBSTATE.OP_POS);
			RETURN;	
		ELSIF nEvent = E_PIEZO_EVENT.MOVE_USER THEN
			ActionMoveUserExecute();
			SetState(E_PIEZO_STATE.OP, E_PIEZO_SUBSTATE.OP_POS);
			RETURN;	
		ELSIF nEvent = E_PIEZO_EVENT.ERRFAULT THEN
			ActionErrExecute();
			SetState(E_PIEZO_STATE.OP, E_PIEZO_SUBSTATE.OP_ERROR);
			RETURN;				
		ELSIF nEvent = E_PIEZO_EVENT.ERRRANGE THEN
			ActionErrExecute();
			SetState(E_PIEZO_STATE.OP, E_PIEZO_SUBSTATE.OP_ERROR);
			RETURN;				
		ELSIF nEvent = E_PIEZO_EVENT.ERRMAXON THEN
			ActionMaxOnFailure();
			SetState(E_PIEZO_STATE.OP, E_PIEZO_SUBSTATE.OP_ERROR);
			RETURN;				
		ELSIF nEvent = E_PIEZO_EVENT.STOP THEN
			ActionStopExecute();
			SetState(E_PIEZO_STATE.OP, E_PIEZO_SUBSTATE.OP_POS);
			RETURN;
		END_IF
		
	E_PIEZO_SUBSTATE.OP_ERROR:			
		IF nEvent = E_PIEZO_EVENT.POS THEN
			ActionPosExecute();
			SetState(E_PIEZO_STATE.OP, E_PIEZO_SUBSTATE.OP_POS);
			RETURN;
		ELSIF nEvent = E_PIEZO_EVENT.HOME THEN
			ActionHomeExecute();
			SetState(E_PIEZO_STATE.OP, E_PIEZO_SUBSTATE.OP_POS);
			RETURN;
		ELSIF nEvent = E_PIEZO_EVENT.AUTO THEN
			ActionAutoExecute();
			SetState(E_PIEZO_STATE.OP, E_PIEZO_SUBSTATE.OP_AUTO);
			RETURN;			
		ELSIF nEvent = E_PIEZO_EVENT.DISABLE THEN
			ActionDisableExecute();
			SetState(E_PIEZO_STATE.NOTOP, E_PIEZO_SUBSTATE.NOTOP_READY);
			RETURN;			
		ELSIF nEvent = E_PIEZO_EVENT.MOVE_BIT THEN
			ActionMoveBitExecute();
			SetState(E_PIEZO_STATE.OP, E_PIEZO_SUBSTATE.OP_POS);
			RETURN;	
		ELSIF nEvent = E_PIEZO_EVENT.MOVE_USER THEN
			ActionMoveUserExecute();
			SetState(E_PIEZO_STATE.OP, E_PIEZO_SUBSTATE.OP_POS);
			RETURN;	
		ELSIF nEvent = E_PIEZO_EVENT.HWOK AND 
			  RefStat.nErrorCode = E_PIEZO_ERROR.HW_NOT_OP THEN
			ActionStopExecute();
			SetState(E_PIEZO_STATE.OP, E_PIEZO_SUBSTATE.OP_POS);
			RETURN;
		ELSIF nEvent = E_PIEZO_EVENT.STOP THEN
			ActionStopExecute();
			RETURN;
		END_IF

		
	END_CASE
	
	(* Transitions from OP state *)
	IF nEvent = E_PIEZO_EVENT.ERRHW THEN
		SetState(E_PIEZO_STATE.OP, E_PIEZO_SUBSTATE.OP_ERROR);
		RETURN;
	ELSIF nEvent = E_PIEZO_EVENT.RESET THEN
		ActionResetExecute();
		SetState(E_PIEZO_STATE.NOTOP, E_PIEZO_SUBSTATE.NOTOP_NOTREADY);
		RETURN;
	END_IF
	
END_CASE

(* 
	"Global" internal transitions valid in any state should go here.
	They do not change the active state configuration. 
	They are evaluated after all the others transitions have been 
	considered.
*) 
IF nEvent = E_PIEZO_EVENT.STOP THEN
	RETURN;
END_IF
END_METHOD

{attribute 'TcRpcEnable':='1'}
METHOD RPC_Auto : INT
VAR_INPUT
END_VAR
// RPC calls are not allowed in Local mode.
IF RefStat.bLocal THEN
	RPC_Auto	:= M_SetRpcStatus(E_PIEZO_RPC_ERROR.LOCAL);
	RETURN;
END_IF

// AUTO command is accepted only if device is in OP state.
IF RefStat.nState <> E_PIEZO_STATE.OP THEN
	RPC_Auto	:= M_SetRpcStatus(E_PIEZO_RPC_ERROR.NOT_OP);
	RETURN;
ELSE
	RefCtrl.nCommand := E_PIEZO_COMMAND.AUTO;
	RefCtrl.bExecute := TRUE;
	
	// Call was successful
	RPC_Auto	:= M_SetRpcStatus(E_PIEZO_RPC_ERROR.OK);
END_IF
END_METHOD

{attribute 'TcRpcEnable':='1'}
METHOD RPC_Disable : INT
VAR_INPUT
END_VAR
// RPC calls are not allowed in Local mode.
IF RefStat.bLocal THEN
	RPC_Disable	:= M_SetRpcStatus(E_PIEZO_RPC_ERROR.LOCAL);
	RETURN;
END_IF

// Disable command is accepted only if device is in OP state.
IF RefStat.nState <> E_PIEZO_STATE.OP THEN
	RPC_Disable	:= M_SetRpcStatus(E_PIEZO_RPC_ERROR.NOT_OP);
	RETURN;
ELSE
	// Set disable command
	RefCtrl.nCommand := E_PIEZO_COMMAND.DISABLE;
	RefCtrl.bExecute := TRUE;
	
	// Call was successful
	RPC_Disable	:= M_SetRpcStatus(E_PIEZO_RPC_ERROR.OK);
END_IF
END_METHOD

{attribute 'TcRpcEnable':='1'}
METHOD RPC_Enable : INT
VAR_INPUT
END_VAR
// RPC calls are not allowed in Local mode.
IF RefStat.bLocal THEN
	RPC_Enable	:= M_SetRpcStatus(E_PIEZO_RPC_ERROR.LOCAL);
	RETURN;
END_IF

// Enable command is accepted only if device is in NOTOP_READY.
IF RefStat.nSubstate <> E_PIEZO_SUBSTATE.NOTOP_READY	THEN
	RPC_Enable	:= M_SetRpcStatus(E_PIEZO_RPC_ERROR.NOT_NOTOP_READY);
	RETURN;
ELSE
	// Set enable command
	RefCtrl.nCommand := E_PIEZO_COMMAND.ENABLE;
	RefCtrl.bExecute := TRUE;

	// Call was successful
	RPC_Enable	:= M_SetRpcStatus(E_PIEZO_RPC_ERROR.OK);
END_IF
END_METHOD

{attribute 'TcRpcEnable':='1'}
METHOD RPC_Home : int
VAR_INPUT
END_VAR
// RPC calls are not allowed in Local mode.
IF RefStat.bLocal THEN
	RPC_Home	:= M_SetRpcStatus(E_PIEZO_RPC_ERROR.LOCAL);
	RETURN;
END_IF

// HOME command is accepted only if device is in OP state.
IF RefStat.nState <> E_PIEZO_STATE.OP THEN
	RPC_Home	:= M_SetRpcStatus(E_PIEZO_RPC_ERROR.NOT_OP);
	RETURN;
ELSE
	RefCtrl.nCommand := E_PIEZO_COMMAND.HOME;
	RefCtrl.bExecute := TRUE;
	
	// Call was successful
	RPC_Home	:= M_SetRpcStatus(E_PIEZO_RPC_ERROR.OK);
END_IF
END_METHOD

{attribute 'TcRpcEnable':='1'}
METHOD RPC_Init : INT
VAR_INPUT
END_VAR
// RPC calls are not allowed in Local mode.
IF RefStat.bLocal THEN
	RPC_Init	:= M_SetRpcStatus(E_PIEZO_RPC_ERROR.LOCAL);
	RETURN;
END_IF

// Init command is accepted only if device is in NOTOP_NOTREADY or ERROR.
IF	RefStat.nSubstate <> E_PIEZO_SUBSTATE.NOTOP_NOTREADY	AND  
	RefStat.nSubstate <> E_PIEZO_SUBSTATE.NOTOP_ERROR		THEN
	RPC_Init	:= M_SetRpcStatus(E_PIEZO_RPC_ERROR.NOT_NOTOP_NOTREADY);
	RETURN;
ELSE
	// Set INIT command
	RefCtrl.nCommand := E_PIEZO_COMMAND.INIT;
	RefCtrl.bExecute := TRUE;
	
	// Call was successful
	RPC_Init	:= M_SetRpcStatus(E_PIEZO_RPC_ERROR.OK);
END_IF
END_METHOD

{attribute 'TcRpcEnable':='1'}
METHOD RPC_MoveBit : INT
VAR_INPUT
	in_nPos1:	INT	:= 0;
	in_nPos2:	INT	:= 0;
	in_nPos3:	INT	:= 0;
END_VAR
VAR
	i:	INT;
END_VAR
// RPC calls are not allowed in Local mode.
IF RefStat.bLocal THEN
	RPC_MoveBit	:= M_SetRpcStatus(E_PIEZO_RPC_ERROR.LOCAL);
	RETURN;
END_IF

// MOVE_BIT command is accepted only if device is in OP state.
IF RefStat.nState <> E_PIEZO_STATE.OP THEN
	RPC_MoveBit	:= M_SetRpcStatus(E_PIEZO_RPC_ERROR.NOT_OP);
	RETURN;
ELSE
	// Copy set positions into ctrl structure
	RefCtrl.nPosBit[0].nValue	:= in_nPos1;
	RefCtrl.nPosBit[1].nValue	:= in_nPos2;
	RefCtrl.nPosBit[2].nValue	:= in_nPos3;

	// Check if the set positions are inside the allowed range
	FOR i:=0 TO RefCfg.nNumAxes-1 DO
		IF NOT M_CheckRangeBit(nIndex:= i, nVal:= RefCtrl.nPosBit[i].nValue) THEN
			M_LogEventError('Set bit value out of range');
			RPC_MoveBit	:= M_SetRpcStatus(E_PIEZO_RPC_ERROR.MOVING_BIT);
			RETURN;
		END_IF
	END_FOR

	// Set MOVE_BIT command
	RefCtrl.nCommand := E_PIEZO_COMMAND.MOVE_BIT;
	RefCtrl.bExecute := TRUE;
	
	// Call was successful
	RPC_MoveBit	:= M_SetRpcStatus(E_PIEZO_RPC_ERROR.OK);
END_IF
END_METHOD

{attribute 'TcRpcEnable':='1'}
METHOD RPC_MoveUser : INT
VAR_INPUT
	in_lrPos1:	LREAL	:= 0;
	in_lrPos2:	LREAL	:= 0;
	in_lrPos3:	LREAL	:= 0;
END_VAR
VAR
	i:	INT;
END_VAR
// RPC calls are not allowed in Local mode.
IF RefStat.bLocal THEN
	RPC_MoveUser	:= M_SetRpcStatus(E_PIEZO_RPC_ERROR.LOCAL);
	RETURN;
END_IF

// MOVE_USER command is accepted only if device is in OP state.
IF RefStat.nState <> E_PIEZO_STATE.OP THEN
	RPC_MoveUser	:= M_SetRpcStatus(E_PIEZO_RPC_ERROR.NOT_OP);
	RETURN;
ELSE
	// Copy set positions into ctrl structure
	RefCtrl.lrPosUser[0].lrValue	:= in_lrPos1;
	RefCtrl.lrPosUser[1].lrValue	:= in_lrPos2;
	RefCtrl.lrPosUser[2].lrValue	:= in_lrPos3;

	// Check if the set positions are inside the allowed range.
	FOR i:=0 TO RefCfg.nNumAxes-1 DO
		IF NOT M_CheckRangeUser(nIndex:= i, lrVal:= RefCtrl.lrPosUser[i].lrValue) THEN
			M_LogEventError('Set User value out of range');
			RPC_MoveUser	:= M_SetRpcStatus(E_PIEZO_RPC_ERROR.MOVING_USER);
			RETURN;
		END_IF
	END_FOR


	// Set MOVE_USER command
	RefCtrl.nCommand := E_PIEZO_COMMAND.MOVE_USER;
	RefCtrl.bExecute := TRUE;
	
	// Call was successful
	RPC_MoveUser	:= M_SetRpcStatus(E_PIEZO_RPC_ERROR.OK);
END_IF
END_METHOD

{attribute 'TcRpcEnable':='1'}
METHOD RPC_Pos : INT
VAR_INPUT
END_VAR
// RPC calls are not allowed in Local mode.
IF RefStat.bLocal THEN
	RPC_Pos	:= M_SetRpcStatus(E_PIEZO_RPC_ERROR.LOCAL);
	RETURN;
END_IF

// POS command is accepted only if device is in OP state.
IF RefStat.nState <> E_PIEZO_STATE.OP THEN
	RPC_Pos	:= M_SetRpcStatus(E_PIEZO_RPC_ERROR.NOT_OP);
	RETURN;
ELSE
	RefCtrl.nCommand := E_PIEZO_COMMAND.POS;
	RefCtrl.bExecute := TRUE;
	
	// Call was successful
	RPC_Pos	:= M_SetRpcStatus(E_PIEZO_RPC_ERROR.OK);
END_IF
END_METHOD

{attribute 'TcRpcEnable':='1'}
METHOD RPC_Reset : INT
VAR_INPUT
END_VAR
// RPC calls are not allowed in Local mode.
IF RefStat.bLocal THEN
	RPC_Reset	:= M_SetRpcStatus(E_PIEZO_RPC_ERROR.LOCAL);
	RETURN;
END_IF

RefCtrl.nCommand := E_PIEZO_COMMAND.RESET;
RefCtrl.bExecute := TRUE;

// Call was successful
RPC_Reset	:= M_SetRpcStatus(E_PIEZO_RPC_ERROR.OK);
END_METHOD

{attribute 'TcRpcEnable':='1'}
METHOD RPC_SetDebug : INT
VAR_INPUT
	in_bDebug:	BOOL 	:= FALSE;		// If TRUE, activate event logging of Debug type
END_VAR
// Enable/disable Debugging
RefCfg.bDebug	:= in_bDebug;

// Call was successful
RPC_SetDebug	:= M_SetRpcStatus(E_PIEZO_RPC_ERROR.OK);
END_METHOD

{attribute 'TcRpcEnable':='1'}
METHOD RPC_SetLog : INT
VAR_INPUT
	in_bLog:	BOOL 	:= FALSE;		// If TRUE, activate event logging
END_VAR
// Enable/disable Logging
RefCfg.bLog	:= in_bLog;

// Call was successful
RPC_SetLog	:= M_SetRpcStatus(E_PIEZO_RPC_ERROR.OK);
END_METHOD

{attribute 'TcRpcEnable':='1'}
METHOD RPC_Stop : INT
VAR_INPUT
END_VAR
// RPC calls are not allowed in Local mode.
IF RefStat.bLocal THEN
	RPC_Stop	:= M_SetRpcStatus(E_PIEZO_RPC_ERROR.LOCAL);
	RETURN;
END_IF

RefCtrl.nCommand := E_PIEZO_COMMAND.STOP;
RefCtrl.bExecute := TRUE;

// Call was successful
RPC_Stop	:= M_SetRpcStatus(E_PIEZO_RPC_ERROR.OK);
END_METHOD

METHOD SetAction
VAR_INPUT
	actionName:		STRING;
END_VAR


RefStat.sActionDesc := actionName;
END_METHOD

METHOD SetEvent
VAR_INPUT
	nEventId:			DINT;
END_VAR

nEvent := nEventId;

CASE nEventId OF
	E_PIEZO_EVENT.NONE:
		RefStat.sEventDesc := '';
		RETURN;
		
	E_PIEZO_EVENT.RESET:
		RefStat.sEventDesc := 'CMD RESET';
		RETURN;
	
	E_PIEZO_EVENT.INIT:
		RefStat.sEventDesc := 'CMD INIT';
		RETURN;

	E_PIEZO_EVENT.STOP:
		RefStat.sEventDesc := 'CMD STOP';
		RETURN;

	E_PIEZO_EVENT.ENABLE:
		RefStat.sEventDesc := 'CMD ENABLE';
		RETURN;

	E_PIEZO_EVENT.DISABLE:
		RefStat.sEventDesc := 'CMD DISABLE';
		RETURN;

	E_PIEZO_EVENT.AUTO:
		RefStat.sEventDesc := 'CMD AUTO';
		RETURN;

	E_PIEZO_EVENT.POS:
		RefStat.sEventDesc := 'CMD POS';
		RETURN;
	
	E_PIEZO_EVENT.HOME:
		RefStat.sEventDesc := 'CMD HOME';
		RETURN;
	
	E_PIEZO_EVENT.MOVE_BIT:
		RefStat.sEventDesc := 'CMD MOVE BIT';
		RETURN;
	
	E_PIEZO_EVENT.MOVE_USER:
		RefStat.sEventDesc := 'CMD MOVE USER';
		RETURN;
	
	(* events corresponding to internal events *)
	E_PIEZO_EVENT.HWOK:
		RefStat.sEventDesc := 'SIG HWOK';
		RETURN;

	E_PIEZO_EVENT.ERRHW:
		RefStat.sEventDesc := 'INT ERRHW';
		RETURN;

	E_PIEZO_EVENT.ERRRANGE:
		RefStat.sEventDesc := 'INT ERRRANGE';
		RETURN;

	E_PIEZO_EVENT.ERRMAXON:
		RefStat.sEventDesc := 'INT ERRMAXON';
		RETURN;

	E_PIEZO_EVENT.ERRFAULT:	
		RefStat.sEventDesc := 'INT ERRFAULT';
		RETURN;

	E_PIEZO_EVENT.ERRINIT:
		RefStat.sEventDesc := 'INT ERRINIT';
		RETURN;

	E_PIEZO_EVENT.ERRDISABLE:
		RefStat.sEventDesc := 'INT ERRDISABLE';
		RETURN;
ELSE
	(* INTERNAL ERROR *)
	RefStat.sEventDesc := 'UNKNOWN EVENT';
	RETURN;
END_CASE
END_METHOD

METHOD SetHwStatus
VAR_INPUT
	hwStatus:	E_PIEZO_HW_STATUS;
END_VAR
RefStat.nHwStatus	:= hwStatus;

CASE hwStatus OF
	E_PIEZO_HW_STATUS.UNKNOWN:
		RefStat.sHwStatus	:= 'UNKNOWN';
	E_PIEZO_HW_STATUS.ERROR:
		RefStat.sHwStatus	:= 'ERROR';
	E_PIEZO_HW_STATUS.ZERO:
		RefStat.sHwStatus	:= 'ZERO';
	E_PIEZO_HW_STATUS.HOME:
		RefStat.sHwStatus	:= 'HOME';
	E_PIEZO_HW_STATUS.POS:
		RefStat.sHwStatus	:= 'POS';
	E_PIEZO_HW_STATUS.AUTO:
		RefStat.sHwStatus	:= 'AUTO';

END_CASE
END_METHOD

METHOD SetLastCommand
VAR_INPUT
	cmd:	E_PIEZO_COMMAND;
END_VAR
RefStat.nLastCommand	:= cmd;

CASE cmd OF
	E_PIEZO_COMMAND.RESET:
		RefStat.sLastCommand	:= 'RESET';
	E_PIEZO_COMMAND.INIT:
		RefStat.sLastCommand	:= 'INIT';
	E_PIEZO_COMMAND.STOP:
		RefStat.sLastCommand	:= 'STOP';
	E_PIEZO_COMMAND.ENABLE:
		RefStat.sLastCommand	:= 'ENABLE';
	E_PIEZO_COMMAND.DISABLE:
		RefStat.sLastCommand	:= 'DISABLE';
	E_PIEZO_COMMAND.AUTO:
		RefStat.sLastCommand	:= 'AUTO';
	E_PIEZO_COMMAND.POS:
		RefStat.sLastCommand	:= 'POS';
	E_PIEZO_COMMAND.HOME:
		RefStat.sLastCommand	:= 'HOME';
ELSE
		RefStat.sLastCommand	:= 'NONE';
END_CASE;
END_METHOD

METHOD SetState
VAR_INPUT
	nState:			E_PIEZO_STATE;
	nSubstate:		E_PIEZO_SUBSTATE;
END_VAR
(* 
	Update State Machine active state configuration.

	ToDo: support initial pseudo state/substate.
*)

IF nState <> E_PIEZO_STATE.NONE THEN
	RefStat.nState	:= nState;
END_IF
IF nSubstate <> E_PIEZO_SUBSTATE.NONE THEN
	RefStat.nSubstate	:= nSubstate;
END_IF

(* Update active state configuration description *)

IF nState = E_PIEZO_STATE.NOTOP THEN
	RefStat.sState	:= 'NOT OP';
ELSIF nState = E_PIEZO_STATE.OP THEN
	RefStat.sState	:= 'OPERATIONAL';
END_IF

IF nSubstate = E_PIEZO_SUBSTATE.NOTOP_NOTREADY THEN
	RefStat.sSubstate	:= 'NOT READY';
ELSIF nSubstate = E_PIEZO_SUBSTATE.NOTOP_READY THEN
	RefStat.sSubstate	:= 'READY';
ELSIF nSubstate = E_PIEZO_SUBSTATE.NOTOP_ERROR THEN
	RefStat.sSubstate	:= 'ERROR';
ELSIF nSubstate = E_PIEZO_SUBSTATE.OP_POS THEN
	RefStat.sSubstate	:= 'POS';
ELSIF nSubstate = E_PIEZO_SUBSTATE.OP_AUTO THEN
	RefStat.sSubstate	:= 'AUTO';
ELSIF nSubstate = E_PIEZO_SUBSTATE.OP_ERROR THEN
	RefStat.sSubstate	:= 'ERROR';
ELSE
	RefStat.sSubstate	:= '';
END_IF


//SetState	:= TRUE;
END_METHOD

METHOD SetStatus
VAR_INPUT
	nErrorCode:	E_PIEZO_ERROR;
	sErrorText:	STRING;
END_VAR
RefStat.nErrorCode 	:= nErrorCode;
RefStat.sErrorText 	:= sErrorText;

IF nErrorCode <> E_PIEZO_ERROR.OK THEN
	RefStat.sStatus	:= 'ERROR';
	RefStat.nStatus	:= E_PIEZO_STATUS.ERROR;
ELSE
	RefStat.sStatus	:= 'OK';
	RefStat.nStatus	:= E_PIEZO_STATUS.OK;
END_IF
END_METHOD

END_FUNCTION_BLOCK

// POUs/FB_SIM_PIEZO
// Simulator that generate sine wave error and
// generate outputs by adding these errors to Piezo outputs (SIM inputs).
FUNCTION_BLOCK FB_SIM_PIEZO
VAR_OUTPUT
END_VAR
VAR
	{attribute 'OPC.UA.DA':='1'}
	cfg:			T_SIM_PIEZO_CFG;		(* ActiveLow configuration for each signal *)

	{attribute 'OPC.UA.DA':='0'}
	nCouplerState:	UINT := 8;       // normal coupler state
	
	{attribute 'OPC.UA.DA':='0'}
	i_nSignal	AT %I*:	ARRAY [0..2] OF INT;			//	Input signals to be linked to Piezo outputs

	{attribute 'OPC.UA.DA':='0'}
	q_nSignal	AT %Q*:	ARRAY [0..2] OF INT;			//	Simulated output signal to be linked to Piezo inputs
	{attribute 'OPC.UA.DA':='0'}
	q_nCouplerState AT %Q*:		UINT := 8;
	
	{attribute 'OPC.UA.DA':='0'}
	timer:			TON;
	
	{attribute 'OPC.UA.DA':='0'}
	initialised:	BOOL := FALSE;		// Used to start timer for the first time
	
	{attribute 'OPC.UA.DA':='0'}
	i:	INT;

END_VAR
VAR_TEMP
	t1:	LREAL;
	t2:	LREAL;
	t3:	LREAL;
	t4:	LREAL;
END_VAR

// Check possible devision by zero
IF cfg.nSignalCycle = 0 THEN
	cfg.nSignalCycle	:= 1000;
END_IF

IF NOT initialised THEN
	initialised := TRUE;
	
	// Start timer for signal=FALSE
	timer(IN:=FALSE);
	timer(IN:=TRUE, PT:=UDINT_TO_TIME(cfg.nSignalCycle));
	RETURN;
END_IF

// Execute timer
// The timer is actually used just for the 'angle' for the sin().
// Angle = ET / PT * 2PI
timer();

// If the timer expired, just restart it
IF timer.Q THEN
		timer(IN:=FALSE);
		timer(IN:=TRUE, PT:=UDINT_TO_TIME(cfg.nSignalCycle));
END_IF

// Set the output
t1	:= TIME_TO_LREAL(timer.ET);
t2	:= TIME_TO_LREAL(timer.PT);
t3	:= t1 / t2 * 2 * 3.14;
t4	:= cfg.nMaxError * SIN(t3);

// Set outputs by adding calculated error to Piezo outputs (SIM inputs)
FOR i:=0 TO 2 DO
	q_nSignal[i] := i_nSignal[i] + LREAL_TO_INT(t4);	
END_FOR

q_nCouplerState := nCouplerState;

{attribute 'TcRpcEnable':='1'}
METHOD RPC_ResetConfig : INT
VAR_INPUT
END_VAR
nCouplerState		:= 8;
cfg.nMaxError		:= 0;
cfg.nSignalCycle	:= 10000;

RPC_ResetConfig	:= 0;
END_METHOD

{attribute 'TcRpcEnable':='1'}
METHOD RPC_SetCouplerState : INT
VAR_INPUT
	nValue:	UINT;	// Coupler State; 8 - OPERATIONAL, anything else - NON OP
END_VAR
nCouplerState	:= nValue;

RPC_SetCouplerState	:= 0;
END_METHOD

{attribute 'TcRpcEnable':='1'}
METHOD RPC_SetMaxError : INT
VAR_INPUT
	nMaxError:		INT;	// Maximal Simulated feedback error [bit]
	nSignalCycle:	UDINT;	// Period for complete sine wave error cycle [msec] 
END_VAR
cfg.nMaxError		:= nMaxError;
cfg.nSignalCycle	:= nSignalCycle;

RPC_SetMaxError	:= 0;
END_METHOD

END_FUNCTION_BLOCK

// POUs/MAIN
PROGRAM MAIN
VAR
	
	{attribute 'OPC.UA.DA':='1'}
	Piezo001:		FB_PIEZO_EXAMPLE;	// Piezo #1
	{attribute 'OPC.UA.DA':='1'}
	Piezo002:		FB_PIEZO_EXAMPLE;	// Piezo #2
	
	{attribute 'OPC.UA.DA':='1'}
	SIM_Piezo001:	FB_SIM_PIEZO;		// Simulator for Piezo #1 (if simulated)
	{attribute 'OPC.UA.DA':='1'}
	SIM_Piezo002:	FB_SIM_PIEZO;		// Simulator for Piezo #2 (always simulated)

END_VAR

Piezo001(in_sName:='Piezo001', in_nNumAxes:=3);

Piezo002(in_sName:='Piezo002', in_nNumAxes:=3);

SIM_Piezo001();
SIM_Piezo002();

END_PROGRAM

// VISUs/Templates/GUI_TEMPLATE_PIEZO
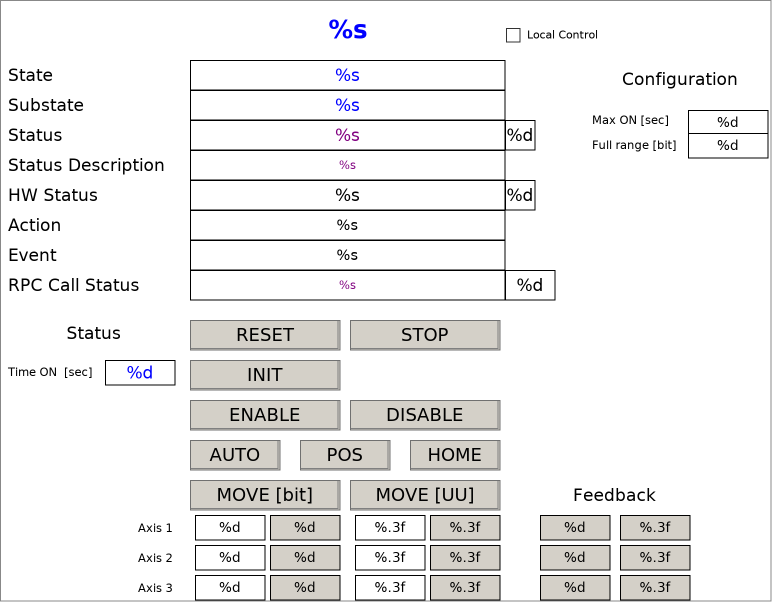
VISUALIZATION GUI_TEMPLATE_PIEZO  // 772x602
VAR_IN_OUT
	m_Instance:	FB_PIEZO_BASE;
END_VAR
    Rectangle (190,60 315x30), "%s", text variable: m_Instance.stat.sState
    Rectangle (190,90 315x30), "%s", text variable: m_Instance.stat.sSubstate
    Button (190,320 150x30), "RESET", input disabled if: (m_Instance.stat.bLocal = FALSE) <> 0
        OnMouseDown: execute { m_Instance.ctrl.nCommand := E_PIEZO_COMMAND.RESET; m_Instance.ctrl.bExecute := TRUE; }
    Button (190,360 150x30), "INIT", input disabled if: (m_Instance.stat.bLocal = FALSE) <> 0
        OnMouseDown: execute { m_Instance.ctrl.nCommand := E_PIEZO_COMMAND.INIT; m_Instance.ctrl.bExecute := TRUE; }
    Button (350,320 150x30), "STOP", input disabled if: (m_Instance.stat.bLocal = FALSE) <> 0
        OnMouseDown: execute { m_Instance.ctrl.nCommand := E_PIEZO_COMMAND.STOP; m_Instance.ctrl.bExecute := TRUE; }
    Button (190,400 150x30), "ENABLE", input disabled if: (m_Instance.stat.bLocal = FALSE) <> 0
        OnMouseDown: execute { m_Instance.ctrl.nCommand := E_PIEZO_COMMAND.ENABLE; m_Instance.ctrl.bExecute := TRUE; }
    Button (350,400 150x30), "DISABLE", input disabled if: (m_Instance.stat.bLocal = FALSE) <> 0
        OnMouseDown: execute { m_Instance.ctrl.nCommand := E_PIEZO_COMMAND.DISABLE; m_Instance.ctrl.bExecute := TRUE; }
    Button (190,440 90x30), "AUTO", tooltip "Start AUTO mode", input disabled if: (m_Instance.stat.bLocal = FALSE) <> 0
        OnMouseDown: execute { m_Instance.ctrl.nCommand := E_PIEZO_COMMAND.AUTO; m_Instance.ctrl.bExecute := TRUE; }
    Button (300,440 90x30), "POS", tooltip "Stop AUTO mode, if running. Keep piezos where they are.", input disabled if: (m_Instance.stat.bLocal = FALSE) <> 0
        OnMouseDown: execute { m_Instance.ctrl.nCommand := E_PIEZO_COMMAND.POS; m_Instance.ctrl.bExecute := TRUE; }
    Rectangle (5,60 180x30), "State"
    Rectangle (5,90 180x30), "Substate"
    Rectangle (190,120 315x30), "%s", text variable: m_Instance.stat.sStatus
    Rectangle (190,150 315x30), "%s", text variable: m_Instance.stat.sErrorText
    Rectangle (5,120 180x30), "Status"
    Rectangle (5,150 180x30), "Status Description"
    Rectangle (190,210 315x30), "%s", text variable: m_Instance.stat.sActionDesc
    Rectangle (190,240 315x30), "%s", text variable: m_Instance.stat.sEventDesc
    Rectangle (190,180 315x30), "%s", text variable: m_Instance.stat.sHwStatus
    Rectangle (5,180 180x30), "HW Status"
    Rectangle (505,180 30x30), "%d", tooltip "HW Status Index", text variable: m_Instance.stat.nHwStatus
    Rectangle (5,210 180x30), "Action"
    Rectangle (5,240 180x30), "Event"
    Rectangle (232,12 232x35), "%s", text variable: m_Instance.cfg.sName
    Rectangle (590,64 180x30), "Configuration"
    Rectangle (589,110 155x20), "Max ON [sec]"
    Rectangle (589,135 155x20), "Full range [bit]"
    Rectangle (688,110 80x25), "%d", tooltip "Maximum allowed time for lamp to be ON [sec] (>=0). Zero means no limit.", text variable: m_Instance.cfg.nMaxOn, input disabled if: (m_Instance.stat.bLocal = FALSE) <> 0
        OnMouseDown: write the text variable via Default, min 0
    Rectangle (688,133 80x25), "%d", tooltip "Full range of A/D converter controlling the intensity [bit]. Examples: 12 bit A/D = 4095 15 bit A/D = 32767 16 bit A/D = 65535", text variable: m_Instance.cfg.nFullRange[0].nValue, input disabled if: (m_Instance.stat.bLocal = FALSE) <> 0
        OnMouseDown: write the text variable via Default, min 0
    Checkbox (504,20 116x30), "Local Control", variable: m_Instance.stat.bLocal
    Rectangle (48,318 92x30), "Status"
    Rectangle (105,360 70x25), "%d", tooltip "Time since last ON command [sec]. Updated only if MaxON > 0.", text variable: m_Instance.stat.nTimeOn
    Rectangle (5,357 95x30), "Time ON [sec]"
    Rectangle (505,120 30x30), "%d", text variable: m_Instance.stat.nStatus
    Button (190,480 150x30), "MOVE [bit]", input disabled if: (m_Instance.stat.bLocal = FALSE) <> 0
        OnMouseDown: execute { m_Instance.ctrl.nCommand := E_PIEZO_COMMAND.MOVE_BIT; m_Instance.ctrl.bExecute := TRUE; }
    Rectangle (195,515 70x25), "%d", tooltip "Axis 1 Set Value [bit]", text variable: m_Instance.ctrl.nPosBit[0].nValue, input disabled if: (m_Instance.stat.bLocal = FALSE) <> 0
        OnMouseDown: write the text variable via Default
    Rectangle (195,545 70x25), "%d", tooltip "Axis 2 Set Value [bit]", text variable: m_Instance.ctrl.nPosBit[1].nValue, input disabled if: (m_Instance.stat.bLocal = FALSE) <> 0
        OnMouseDown: write the text variable via Default
    Button (350,480 150x30), "MOVE [UU]", input disabled if: (m_Instance.stat.bLocal = FALSE) <> 0
        OnMouseDown: execute { m_Instance.ctrl.nCommand := E_PIEZO_COMMAND.MOVE_USER; m_Instance.ctrl.bExecute := TRUE; }
    Rectangle (355,515 70x25), "%.3f", tooltip "Axis 1 Set position [UU]", text variable: m_Instance.ctrl.lrPosUser[0].lrValue, input disabled if: (m_Instance.stat.bLocal = FALSE) <> 0
        OnMouseDown: write the text variable via Default
    Rectangle (355,545 70x25), "%.3f", tooltip "Axis 2 Set position [UU]", text variable: m_Instance.ctrl.lrPosUser[1].lrValue, input disabled if: (m_Instance.stat.bLocal = FALSE) <> 0
        OnMouseDown: write the text variable via Default
    Rectangle (270,515 70x25), "%d", tooltip "Axis 1 Actual Output [bit]", text variable: m_Instance.q_nCtrl[0], input disabled if: TRUE
        OnMouseDown: write the text variable via Default, min 0
    Rectangle (270,545 70x25), "%d", tooltip "Axis 2 Actual Output [bit]", text variable: m_Instance.q_nCtrl[1], input disabled if: TRUE
        OnMouseDown: write the text variable via Default, min 0
    Rectangle (430,515 70x25), "%.3f", tooltip "Axis 1 Actual Output [UU]", text variable: m_Instance.stat.lrSetPosUsr[0].lrValue, input disabled if: TRUE
        OnMouseDown: write the text variable via Default, min 0
    Rectangle (430,545 70x25), "%.3f", tooltip "Axis 2 Actual Output [UU]", text variable: m_Instance.stat.lrSetPosUsr[1].lrValue, input disabled if: TRUE
        OnMouseDown: write the text variable via Default, min 0
    Button (410,440 90x30), "HOME", tooltip "Home piezos", input disabled if: (m_Instance.stat.bLocal = FALSE) <> 0
        OnMouseDown: execute { m_Instance.ctrl.nCommand := E_PIEZO_COMMAND.HOME; m_Instance.ctrl.bExecute := TRUE; }
    Rectangle (195,575 70x25), "%d", tooltip "Axis 3 Set Value [bit]", text variable: m_Instance.ctrl.nPosBit[2].nValue, input disabled if: (m_Instance.stat.bLocal = FALSE) <> 0
        OnMouseDown: write the text variable via Default
    Rectangle (355,575 70x25), "%.3f", tooltip "Axis 3 Set position [UU]", text variable: m_Instance.ctrl.lrPosUser[2].lrValue, input disabled if: (m_Instance.stat.bLocal = FALSE) <> 0
        OnMouseDown: write the text variable via Default
    Rectangle (270,575 70x25), "%d", tooltip "Axis 3 Actual Output [bit]", text variable: m_Instance.q_nCtrl[2], input disabled if: TRUE
        OnMouseDown: write the text variable via Default, min 0
    Rectangle (430,575 70x25), "%.3f", tooltip "Axis 3 Actual Output [UU]", text variable: m_Instance.stat.lrSetPosUsr[2].lrValue, input disabled if: TRUE
        OnMouseDown: write the text variable via Default, min 0
    Rectangle (135,518 55x20), "Axis 1"
    Rectangle (135,548 55x20), "Axis 2"
    Rectangle (135,578 55x20), "Axis 3"
    Rectangle (190,270 315x30), "%s", text variable: m_Instance.stat.sRpcErrorText
    Rectangle (5,270 180x30), "RPC Call Status"
    Rectangle (505,270 50x30), "%d", tooltip "RPC Error Code 0 - OK", text variable: m_Instance.stat.nRpcErrorCode
    Rectangle (540,515 70x25), "%d", tooltip "Axis 1 Feedback [bit]", text variable: m_Instance.stat.nActPosBit[0].nValue, input disabled if: TRUE
        OnMouseDown: write the text variable via Default, min 0
    Rectangle (550,480 129x30), "Feedback"
    Rectangle (620,515 70x25), "%.3f", tooltip "Axis 1 Feedback [UU]", text variable: m_Instance.stat.lrActPosUsr[0].lrValue, input disabled if: TRUE
        OnMouseDown: write the text variable via Default, min 0
    Rectangle (540,545 70x25), "%d", tooltip "Axis 2 Feedback [bit]", text variable: m_Instance.stat.nActPosBit[1].nValue, input disabled if: TRUE
        OnMouseDown: write the text variable via Default, min 0
    Rectangle (620,545 70x25), "%.3f", tooltip "Axis 2 Feedback [UU]", text variable: m_Instance.stat.lrActPosUsr[1].lrValue, input disabled if: TRUE
        OnMouseDown: write the text variable via Default, min 0
    Rectangle (540,575 70x25), "%d", tooltip "Axis 3 Feedback [bit]", text variable: m_Instance.stat.nActPosBit[2].nValue, input disabled if: TRUE
        OnMouseDown: write the text variable via Default, min 0
    Rectangle (620,575 70x25), "%.3f", tooltip "Axis 3 Feedback [UU]", text variable: m_Instance.stat.lrActPosUsr[2].lrValue, input disabled if: TRUE
        OnMouseDown: write the text variable via Default, min 0
END_VISUALIZATION

// VISUs/GUI_Piezo001
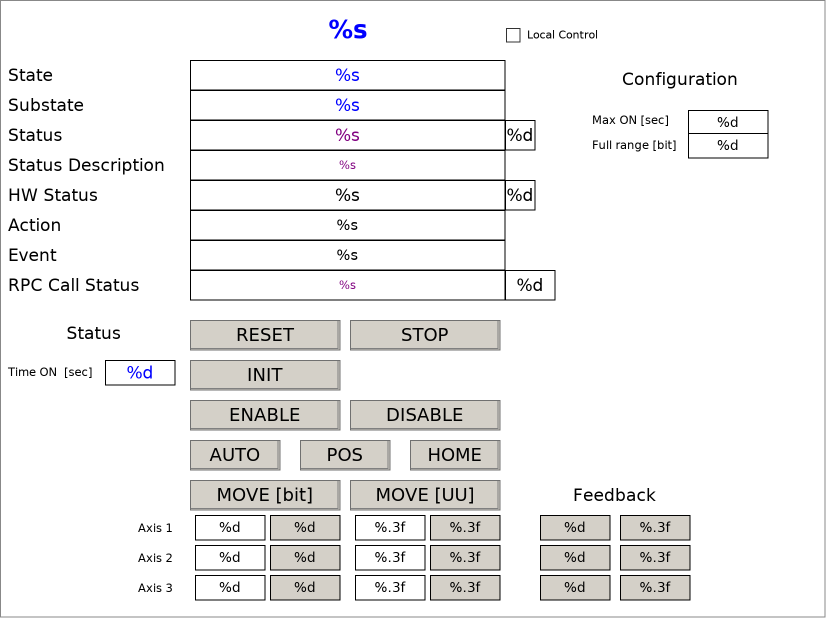
VISUALIZATION GUI_Piezo001  // 826x618
    Frame (0,0 824x616)
        shows GUI_TEMPLATE_PIEZO(m_Instance := MAIN.Piezo001)
END_VISUALIZATION

// VISUs/GUI_Piezo002
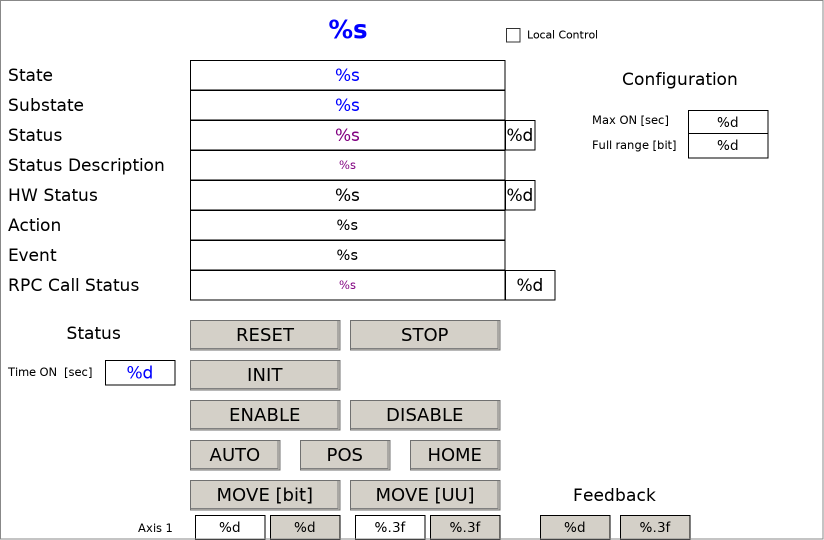
VISUALIZATION GUI_Piezo002  // 824x540
    Frame (0,0 824x540)
        shows GUI_TEMPLATE_PIEZO(m_Instance := MAIN.Piezo002)
END_VISUALIZATION
